# B&R Automation Studio project NAINV104C00R8L515F00 (part 13)

#### Act_EntP0940Disp.st
```iecst
ACTION Act_EntP0940Disp:

	//Access Address
	p_tyC0002FullMask ACCESS ADR(tyP0940CommCtrl.tyFullMaskHide);

	p_tyC0005Main ACCESS ADR(tyCommon.tyMain);

	p_tyC0007Notif ACCESS ADR(tyCommon.tyNotif);

	p_tyC0008MsgBox ACCESS ADR(tyP0940CommCtrl.tyMsgBoxHide);

	p_tyC0009Info ACCESS ADR(tyCommon.tyInfo);

	p_tyC0011Loading ACCESS ADR(tyCommon.tyLoading);

	p_tyP0940CommCtrlUSSMEMA ACCESS ADR(tyP0940CommCtrl.tyUSSMEMA);

	p_tyP0940CommCtrlDSSMEMA ACCESS ADR(tyP0940CommCtrl.tyDSSMEMA);

	p_tyP0940CommCtrlUSSMEMA2 ACCESS ADR(tyP0940CommCtrl.tyUSSMEMA2);

	//Display - Upstream
	fUIInRtStatOff(ADR(tyP0940CommCtrl.tyUSSMEMA.tyLyr.uiRtStat));

	IF p_tyMcParamCurr.tyUSCommSMEMA.eSelection = SMEMASelIPC9851Ext THEN
		fUIInRtStatOff(ADR(tyP0940CommCtrl.tyUSSMEMA.tyBtnUBAStat.uiRtStat));

		IF p_tyMcParamCurr.tyUSCommSMEMA.bStatSigSetGd = TRUE THEN
			tyP0940CommCtrl.tyUSSMEMA.tyBtnUBAStat.usiTxtIdx	:= 1;
		ELSE
			tyP0940CommCtrl.tyUSSMEMA.tyBtnUBAStat.usiTxtIdx	:= 2;
		END_IF
	ELSE
		fUIInRtStatHide(ADR(tyP0940CommCtrl.tyUSSMEMA.tyBtnUBAStat.uiRtStat));
	END_IF

	//Display - Upstream 2
	fUIInRtStatOff(ADR(tyP0940CommCtrl.tyUSSMEMA2.tyLyr.uiRtStat));

	IF p_tyMcParamCurr.tyUSCommSMEMA2.eSelection = SMEMASelIPC9851Ext THEN
		fUIInRtStatOff(ADR(tyP0940CommCtrl.tyUSSMEMA2.tyBtnUBAStat.uiRtStat));

		IF p_tyMcParamCurr.tyUSCommSMEMA2.bStatSigSetGd = TRUE THEN
			tyP0940CommCtrl.tyUSSMEMA2.tyBtnUBAStat.usiTxtIdx	:= 1;
		ELSE
			tyP0940CommCtrl.tyUSSMEMA2.tyBtnUBAStat.usiTxtIdx	:= 2;
		END_IF
	ELSE
		fUIInRtStatHide(ADR(tyP0940CommCtrl.tyUSSMEMA2.tyBtnUBAStat.uiRtStat));
	END_IF

	//Display - Downstream
	fUIInRtStatOff(ADR(tyP0940CommCtrl.tyDSSMEMA.tyLyr.uiRtStat));

	IF p_tyMcParamCurr.tyDSCommSMEMA.eSelection = SMEMASelIPC9851Ext THEN
		fUIInRtStatOff(ADR(tyP0940CommCtrl.tyDSSMEMA.tyBtnDBAStat.uiRtStat));

		IF p_tyMcParamCurr.tyDSCommSMEMA.bStatSigSetGd = TRUE THEN
			tyP0940CommCtrl.tyDSSMEMA.tyBtnDBAStat.usiTxtIdx	:= 1;
		ELSE
			tyP0940CommCtrl.tyDSSMEMA.tyBtnDBAStat.usiTxtIdx	:= 2;
		END_IF
	ELSE
		fUIInRtStatHide(ADR(tyP0940CommCtrl.tyDSSMEMA.tyBtnDBAStat.uiRtStat));
	END_IF

END_ACTION
```

#### Act_OptP0940FullMask.st
```iecst
ACTION Act_OptP0940FullMask:

	IF eCurrPage = UIP0940CommCtrl THEN

		IF p_tyDI.bEStopSig = FALSE THEN
			p_tyC0002FullMask ACCESS ADR(tyP0940CommCtrl.tyFullMaskEStop);

		ELSIF p_tyDI.bCoverSWSig = FALSE THEN
			p_tyC0002FullMask ACCESS ADR(tyP0940CommCtrl.tyFullMaskCWSig);

		ELSIF p_tyDI.bSafetyRlySig = FALSE THEN
			p_tyC0002FullMask ACCESS ADR(tyP0940CommCtrl.tyFullMaskSafetyRly);

		ELSE
			p_tyC0002FullMask ACCESS ADR(tyP0940CommCtrl.tyFullMaskHide);

		END_IF

	END_IF

END_ACTION
```

#### Act_OptP0940ReadDI.st
```iecst
ACTION Act_OptP0940ReadDI:

	tyP0940CommCtrl.tyUSSMEMA.tyBtnUBA.bValue			:= p_tyDI.bUBA;
	tyP0940CommCtrl.tyUSSMEMA.tyBtnUBAStat.bValue		:= p_tyDI.bUBAStat;

	tyP0940CommCtrl.tyDSSMEMA.tyBtnDSB.bValue			:= p_tyDI.bDSB;

	tyP0940CommCtrl.tyUSSMEMA2.tyBtnUBA.bValue			:= p_tyDI.bUBA2;
	tyP0940CommCtrl.tyUSSMEMA2.tyBtnUBAStat.bValue		:= p_tyDI.bUBAStat2;

END_ACTION
```

#### Act_OptP0940WriteDO.st
```iecst
ACTION Act_OptP0940WriteDO:

	// USB
	IF tyP0940CommCtrl.tyUSSMEMA.tyBtnUSB.bRtCompl = TRUE THEN
		IF tyP0940CommCtrl.tyUSSMEMA.tyBtnUSB.bValue = TRUE THEN
			eUSSMEMAAct	:= SMEMAActSetSig;

			IF p_eUSSMEMAStat = SMEMAActSetSig AND p_eUSSMEMAStatus = Done THEN
				eUSSMEMAAct	:= SMEMAActIdle;

				tyP0940CommCtrl.tyUSSMEMA.tyBtnUSB.bRtCompl	:= FALSE;
			END_IF
		ELSE
			eUSSMEMAAct	:= SMEMAActRstSig;

			IF p_eUSSMEMAStat = SMEMAActRstSig AND p_eUSSMEMAStatus = Done THEN
				eUSSMEMAAct	:= SMEMAActIdle;

				tyP0940CommCtrl.tyUSSMEMA.tyBtnUSB.bRtCompl	:= FALSE;
			END_IF
		END_IF
	END_IF

	// USB2
	IF tyP0940CommCtrl.tyUSSMEMA2.tyBtnUSB.bRtCompl = TRUE THEN
		IF tyP0940CommCtrl.tyUSSMEMA2.tyBtnUSB.bValue = TRUE THEN
			eUSSMEMA2Act	:= SMEMAActSetSig;

			IF p_eUSSMEMA2Stat = SMEMAActSetSig AND p_eUSSMEMA2Status = Done THEN
				eUSSMEMA2Act	:= SMEMAActIdle;

				tyP0940CommCtrl.tyUSSMEMA2.tyBtnUSB.bRtCompl	:= FALSE;
			END_IF
		ELSE
			eUSSMEMA2Act	:= SMEMAActRstSig;

			IF p_eUSSMEMA2Stat = SMEMAActRstSig AND p_eUSSMEMA2Status = Done THEN
				eUSSMEMA2Act	:= SMEMAActIdle;

				tyP0940CommCtrl.tyUSSMEMA2.tyBtnUSB.bRtCompl	:= FALSE;
			END_IF
		END_IF
	END_IF

	// DBA
	IF tyP0940CommCtrl.tyDSSMEMA.tyBtnDBA.bRtCompl = TRUE THEN
		IF tyP0940CommCtrl.tyDSSMEMA.tyBtnDBA.bValue = TRUE THEN
			eDSSMEMAAct	:= SMEMAActSetSig;

			IF p_eDSSMEMAStat = SMEMAActSetSig AND p_eDSSMEMAStatus = Done THEN
				eDSSMEMAAct	:= SMEMAActIdle;

				tyP0940CommCtrl.tyDSSMEMA.tyBtnDBA.bRtCompl	:= FALSE;
			END_IF
		ELSE
			eDSSMEMAAct	:= SMEMAActRstSig;

			IF p_eDSSMEMAStat = SMEMAActRstSig AND p_eDSSMEMAStatus = Done THEN
				eDSSMEMAAct	:= SMEMAActIdle;

				tyP0940CommCtrl.tyDSSMEMA.tyBtnDBA.bRtCompl	:= FALSE;
			END_IF
		END_IF
	END_IF

	// DBA Stat
	IF tyP0940CommCtrl.tyDSSMEMA.tyBtnDBAStat.bRtCompl = TRUE THEN
		IF tyP0940CommCtrl.tyDSSMEMA.tyBtnDBAStat.bValue = TRUE THEN
			eDSSMEMAAct	:= SMEMAActSetStatSig;

			IF p_eDSSMEMAStat = SMEMAActSetStatSig AND p_eDSSMEMAStatus = Done THEN
				eDSSMEMAAct	:= SMEMAActIdle;

				tyP0940CommCtrl.tyDSSMEMA.tyBtnDBAStat.bRtCompl	:= FALSE;
			END_IF
		ELSE
			eDSSMEMAAct	:= SMEMAActRstStatSig;

			IF p_eDSSMEMAStat = SMEMAActRstStatSig AND p_eDSSMEMAStatus = Done THEN
				eDSSMEMAAct	:= SMEMAActIdle;

				tyP0940CommCtrl.tyDSSMEMA.tyBtnDBAStat.bRtCompl	:= FALSE;
			END_IF
		END_IF
	END_IF

END_ACTION
```

#### Act_OptP0940UpdtDat.st
```iecst
ACTION Act_OptP0940UpdtDat:

	//Hermes Comm
	//Upstream
	g_tyP0940CommCtrl.tyHermesUS.tyBitmapHermes.uiMaskRtStat.0		:= tyUSHermesBackgndData.bConnectionOK;
	g_tyP0940CommCtrl.tyHermesUS.tyBtnExecute.uiMaskRtStat.0		:= tyUSHermesBackgndData.bConnectionOK;

	IF tyUSHermesBackgndData.bConnectionOK = FALSE THEN
		g_tyP0940CommCtrl.tyHermesUS.tyTxtStat.usiValueIdx	:= 0;
	ELSIF tyUSHermesBackgndData.bConnectionOK = TRUE THEN
		g_tyP0940CommCtrl.tyHermesUS.tyTxtStat.usiValueIdx	:= 1;
	END_IF

	//LED ON
	g_tyP0940CommCtrl.tyHermesUS.tyBtnChkAlive.bValue				:= tyUSHermesBackgndData.tyHermesAllDataFromUS.tyCheckAlive.bChkAlive;
	g_tyP0940CommCtrl.tyHermesUS.tyBtnServiceDescription.bValue		:= tyUSHermesBackgndData.tyHermesAllDataFromUS.tyServiceDescription.bServiceDescription;
	g_tyP0940CommCtrl.tyHermesUS.tyBtnBrdAvl.bValue					:= tyUSHermesBackgndData.tyHermesAllDataFromUS.tyBoardAvailable.bBrdAvl;
	g_tyP0940CommCtrl.tyHermesUS.tyBtnRevokeBrdAvl.bValue			:= tyUSHermesBackgndData.tyHermesAllDataFromUS.tyRevokeBoardAvailable.bRevokeBrdAvl;
	g_tyP0940CommCtrl.tyHermesUS.tyBtnTransportFinished.bValue		:= tyUSHermesBackgndData.tyHermesAllDataFromUS.tyTransportFinished.bTransportFinished;

	//Downstream
	g_tyP0940CommCtrl.tyHermesDS.tyBitmapHermes.uiMaskRtStat.0		:= tyDSHermesBackgndData.bConnectionOK;
	g_tyP0940CommCtrl.tyHermesDS.tyBtnExecute.uiMaskRtStat.0		:= tyDSHermesBackgndData.bConnectionOK;

	IF tyDSHermesBackgndData.bConnectionOK = FALSE THEN
		g_tyP0940CommCtrl.tyHermesDS.tyTxtStat.usiValueIdx	:= 0;
	ELSIF tyDSHermesBackgndData.bConnectionOK = TRUE THEN
		g_tyP0940CommCtrl.tyHermesDS.tyTxtStat.usiValueIdx	:= 1;
	END_IF

	//LED ON
	g_tyP0940CommCtrl.tyHermesDS.tyBtnChkAlive.bValue				:= tyDSHermesBackgndData.tyHermesAllDataFromDS.tyCheckAlive.bChkAlive;
	g_tyP0940CommCtrl.tyHermesDS.tyBtnServiceDescription.bValue		:= tyDSHermesBackgndData.tyHermesAllDataFromDS.tyServiceDescription.bServiceDescription;
	g_tyP0940CommCtrl.tyHermesDS.tyBtnMcRdy.bValue					:= tyDSHermesBackgndData.tyHermesAllDataFromDS.tyMachineReady.bMcRdy;
	g_tyP0940CommCtrl.tyHermesDS.tyBtnRevokeMcRdy.bValue			:= tyDSHermesBackgndData.tyHermesAllDataFromDS.tyRevokeMachineReady.bRevokeMcRdy;
	g_tyP0940CommCtrl.tyHermesDS.tyBtnStartTransport.bValue			:= tyDSHermesBackgndData.tyHermesAllDataFromDS.tyStartTransport.bStartTransport;
	g_tyP0940CommCtrl.tyHermesDS.tyBtnStopTransport.bValue			:= tyDSHermesBackgndData.tyHermesAllDataFromDS.tyStopTransport.bStopTransport;

END_ACTION
```

#### Act_OptP0940MsgCtrl.st
```iecst
ACTION Act_OptP0940MsgCtrl:

	//Upstream
	IF g_tyP0940CommCtrl.tyHermesUS.tyBtnExecute.bRtCompl = TRUE THEN
		g_tyP0940CommCtrl.tyHermesUS.tyBtnExecute.bRtCompl	:= FALSE;
		g_tyP0940CommCtrl.tyHermesUS.tyBtnExecute.bValue	:= FALSE;

		IF g_tyP0940CommCtrl.tyHermesUS.tyDrpDnMsgList.usiValueIdx = 0 THEN
			tyUSHermesBackgndData.tyHermesAllDataToUS.tyCheckAlive.bChkAlive					:= TRUE;
		ELSIF g_tyP0940CommCtrl.tyHermesUS.tyDrpDnMsgList.usiValueIdx = 1 THEN
			tyUSHermesBackgndData.tyHermesAllDataToUS.tyServiceDescription.bServiceDescription	:= TRUE;
		ELSIF g_tyP0940CommCtrl.tyHermesUS.tyDrpDnMsgList.usiValueIdx = 2 THEN
			tyUSHermesBackgndData.tyHermesAllDataToUS.tyMachineReady.bMcRdy						:= TRUE;
		ELSIF g_tyP0940CommCtrl.tyHermesUS.tyDrpDnMsgList.usiValueIdx = 3 THEN
			tyUSHermesBackgndData.tyHermesAllDataToUS.tyRevokeMachineReady.bRevokeMcRdy			:= TRUE;
		ELSIF g_tyP0940CommCtrl.tyHermesUS.tyDrpDnMsgList.usiValueIdx = 4 THEN
			tyUSHermesBackgndData.tyHermesAllDataToUS.tyStartTransport.bStartTransport			:= TRUE;
		ELSIF g_tyP0940CommCtrl.tyHermesUS.tyDrpDnMsgList.usiValueIdx = 5 THEN
			tyUSHermesBackgndData.tyHermesAllDataToUS.tyStopTransport.bStopTransport			:= TRUE;
		ELSIF g_tyP0940CommCtrl.tyHermesUS.tyDrpDnMsgList.usiValueIdx = 6 THEN
			fbUSHermesBackgnd1.eAct	:= HermesBackgroundActIdle;
		END_IF
	END_IF

	//Downstream
	IF g_tyP0940CommCtrl.tyHermesDS.tyBtnExecute.bRtCompl = TRUE THEN
		g_tyP0940CommCtrl.tyHermesDS.tyBtnExecute.bRtCompl	:= FALSE;
		g_tyP0940CommCtrl.tyHermesDS.tyBtnExecute.bValue	:= FALSE;

		IF g_tyP0940CommCtrl.tyHermesDS.tyDrpDnMsgList.usiValueIdx = 0 THEN
			tyDSHermesBackgndData.tyHermesAllDataToDS.tyCheckAlive.bChkAlive					:= TRUE;
		ELSIF g_tyP0940CommCtrl.tyHermesDS.tyDrpDnMsgList.usiValueIdx = 1 THEN
			tyDSHermesBackgndData.tyHermesAllDataToDS.tyServiceDescription.bServiceDescription	:= TRUE;
		ELSIF g_tyP0940CommCtrl.tyHermesDS.tyDrpDnMsgList.usiValueIdx = 2 THEN
			tyDSHermesBackgndData.tyHermesAllDataToDS.tyBoardAvailable.bBrdAvl					:= TRUE;
		ELSIF g_tyP0940CommCtrl.tyHermesDS.tyDrpDnMsgList.usiValueIdx = 3 THEN
			tyDSHermesBackgndData.tyHermesAllDataToDS.tyRevokeBoardAvailable.bRevokeBrdAvl		:= TRUE;
		ELSIF g_tyP0940CommCtrl.tyHermesDS.tyDrpDnMsgList.usiValueIdx = 4 THEN
			tyDSHermesBackgndData.tyHermesAllDataToDS.tyTransportFinished.bTransportFinished	:= TRUE;
		ELSIF g_tyP0940CommCtrl.tyHermesDS.tyDrpDnMsgList.usiValueIdx = 5 THEN
			fbDSHermesBackgnd1.eAct	:= HermesBackgroundActIdle;
		END_IF
	END_IF

END_ACTION
```

#### Act_OptP0940RstMnl.st
```iecst
ACTION Act_OptP0940RstMnl:

	IF EDGEPOS((bManualMod = FALSE) OR (p_eUSSMEMAStatus = Error OR p_eDSSMEMAStatus = Error)) THEN

		eUSSMEMAAct		:= SMEMAActIdle;
		eDSSMEMAAct		:= SMEMAActIdle;
		eUSSMEMA2Act	:= SMEMAActIdle;

		//SMEMA
		tyP0940CommCtrl.tyUSSMEMA.tyBtnUSB.bValue			:= FALSE;
		tyP0940CommCtrl.tyDSSMEMA.tyBtnDBA.bValue			:= FALSE;
		tyP0940CommCtrl.tyDSSMEMA.tyBtnDBAStat.bValue		:= FALSE;
		tyP0940CommCtrl.tyUSSMEMA2.tyBtnUBA.bValue			:= FALSE;

	END_IF

END_ACTION
```

#### Act_EntP0950Disp.st
```iecst
ACTION Act_EntP0950Disp:

	//Access Address
	p_tyC0005Main ACCESS ADR(tyCommon.tyMain);

	p_tyC0007Notif ACCESS ADR(tyCommon.tyNotif);

	p_tyC0008MsgBox ACCESS ADR(tyP0950Simu.tyMsgBoxHide);

	p_tyC0002FullMask ACCESS ADR (tyP0950Simu.tyFullMaskHide);

	p_tyC0009Info ACCESS ADR(tyCommon.tyInfo);

	p_tyP0950Simu ACCESS ADR(tyP0950Simu.tySimu);

	p_tyC0011Loading ACCESS ADR(tyCommon.tyLoading);

END_ACTION
```

#### Act_OptP0950SimulationMod.st
```iecst
ACTION Act_OptP0950SimulationMod:

	IF p_bSimuStatusRun THEN
		tyP0950Simu.tySimu.tyBtnSimu.bRtLk				:= TRUE;
	ELSE
		tyP0950Simu.tySimu.tyBtnSimu.bRtLk				:= tyP0950Simu.tySimu.tyBtnSimu.bValue;
	END_IF

	IF tyP0950Simu.tySimu.tyBtnSimu.bRtCompl THEN
		tyP0950Simu.tySimu.tyBtnSimu.bRtCompl 			:= FALSE;
		tyP0950Simu.tySimu.tyBtnSimu.bValue	  			:= TRUE;
		tyP0950Simu.tySimu.tyBtnSimu.bRtLk	  			:= TRUE;
	END_IF

END_ACTION
```

#### Act_OptP0950Control.st
```iecst
ACTION Act_OptP0950Control:

	// Error
	IF EDGEPOS(p_bAlarmErr = TRUE AND p_bSimuStatusStop = FALSE) THEN

		tyP0950Simu.tySimu.tyBtnStart.bRtCompl	:= FALSE;
		tyP0950Simu.tySimu.tyBtnStop.bRtCompl	:= FALSE;

		tyP0950Simu.tySimu.tyBtnStart.bValue	:= FALSE;
		tyP0950Simu.tySimu.tyBtnStop.bValue		:= FALSE;

		eSimuAct	:= SimulationsActError;

	ELSE

		IF p_eSimuStat = SimulationsActError AND p_eSimuStatus = Done THEN
			eSimuAct	:= SimulationsActIdle;

			bSimuMod	:= FALSE;

		END_IF

	END_IF

	//Control
	IF tyP0950Simu.tySimu.tyBtnStart.bRtCompl = TRUE THEN
		tyP0950Simu.tySimu.tyBtnStop.bRtCompl	:= FALSE;

		eSimuAct		:= SimulationsActStart;

		bSimuMod		:= TRUE;

		IF p_eSimuStat = SimulationsActStart AND p_eSimuStatus = Done THEN
			eSimuAct	:= SimulationsActIdle;

			tyP0950Simu.tySimu.tyBtnStart.bRtCompl	:= FALSE;

		END_IF

	ELSIF tyP0950Simu.tySimu.tyBtnStop.bRtCompl = TRUE THEN
		tyP0950Simu.tySimu.tyBtnStart.bRtCompl	:= FALSE;

		eSimuAct			:= SimulationsActStop;

		IF p_eSimuStat = SimulationsActStop AND p_eSimuStatus = Done THEN
			eSimuAct		:= SimulationsActIdle;
			bSimuMod		:= FALSE;

			tyP0950Simu.tySimu.tyBtnStop.bRtCompl	:= FALSE;
		END_IF

	END_IF

	// Mask
	IF p_bAlarmErr = TRUE THEN
		fUIInRtStatOff(ADR(tyP0950Simu.tySimu.tyBtnStart.uiMaskRtStat));
		fUIInRtStatOff(ADR(tyP0950Simu.tySimu.tyBtnStop.uiMaskRtStat));

	ELSIF p_bSimuStatusCycleStop = TRUE THEN
		fUIInRtStatHide(ADR(tyP0950Simu.tySimu.tyBtnStart.uiMaskRtStat));
		fUIInRtStatOff(ADR(tyP0950Simu.tySimu.tyBtnStop.uiMaskRtStat));

		fbStopBlinkTm(IN := TRUE);
		IF fbStopBlinkTm.Q = TRUE THEN
			fbStopBlinkTm(IN := FALSE);

			tyP0950Simu.tySimu.tyBtnStart.bValue		:= NOT tyP0950Simu.tySimu.tyBtnStart.bValue;
		END_IF

	ELSIF p_bSimuStatusRun = TRUE THEN
		fUIInRtStatOff(ADR(tyP0950Simu.tySimu.tyBtnStart.uiMaskRtStat));
		fUIInRtStatHide(ADR(tyP0950Simu.tySimu.tyBtnStop.uiMaskRtStat));

	ELSE
		fUIInRtStatHide(ADR(tyP0950Simu.tySimu.tyBtnStart.uiMaskRtStat));
		fUIInRtStatOff(ADR(tyP0950Simu.tySimu.tyBtnStop.uiMaskRtStat));

	END_IF

END_ACTION
```

#### Act_EntP1000Disp.st
```iecst
ACTION Act_EntP1000Disp:

	//Access Address
	p_tyC0005Main ACCESS ADR(tyCommon.tyMain);

	p_tyC0007Notif ACCESS ADR(tyCommon.tyNotif);

	p_tyC0008MsgBox ACCESS ADR(tyP1000Lang.tyMsgBoxHide);

	p_tyC0009Info ACCESS ADR(tyCommon.tyInfo);

	p_tyC0011Loading ACCESS ADR(tyCommon.tyLoading);

	p_tyP1000Lang ACCESS ADR(tyP1000Lang.tyLang);

	//Backup Param
	tyP1000Lang.tyLangBkUp	:= tyP1000Lang.tyLang;

	//Display
	tyP1000Lang.tyLang.tyBtnEnglish.uiRtStat.0		:= NOT (p_tyNtParamCurr.bChinesePrep OR p_tyNtParamCurr.bGemanPrep);
	tyP1000Lang.tyLang.tyBtnChinese.uiRtStat.0		:= NOT (p_tyNtParamCurr.bChinesePrep);
	tyP1000Lang.tyLang.tyBtnGerman.uiRtStat.0		:= NOT (p_tyNtParamCurr.bGemanPrep);

END_ACTION
```

#### Act_ExitP1000.st
```iecst
ACTION Act_ExitP1000:

	eMcParamAct	:= McParamActWrite;

	IF p_eMcParamStat = McParamActWrite AND p_eMcParamStatus = Done THEN
		eMcParamAct	:= McParamActIdle;

		usiChgPage	:= 1;

	ELSIF p_eMcParamStatus = Error THEN
		p_tyC0008MsgBox ACCESS ADR(tyP1000Lang.tyMsgBoxSaveErr);

		IF tyP1000Lang.tyMsgBoxSaveErr.tyBtnNo.bRtCompl = TRUE THEN
			tyP1000Lang.tyMsgBoxSaveErr.tyBtnNo.bRtCompl	:= FALSE;
			tyP1000Lang.tyMsgBoxSaveErr.tyBtnNo.bValue		:= FALSE;

			p_tyC0008MsgBox ACCESS ADR(tyP1000Lang.tyMsgBoxHide);

			//Restore Param
			tyP1000Lang.tyLang				:= tyP1000Lang.tyLangBkUp;
			tyMcParamWr						:= p_tyMcParamCurr;
			tyProperty.tyVisu.usiChgLang	:= p_tyMcParamCurr.usiLang;

			usiChgPage	:= 1;

		END_IF

	END_IF

END_ACTION
```

#### Act_OptP1000SelectLang.st
```iecst
ACTION Act_OptP1000SelectLang:

	// Select English Language
	IF tyP1000Lang.tyLang.tyBtnEnglish.bRtCompl = TRUE THEN
		tyP1000Lang.tyLang.tyBtnEnglish.bRtCompl	:= FALSE;

		tyP1000Lang.tyLang.tyBtnEnglish.bValue		:= TRUE;
		tyP1000Lang.tyLang.tyBtnGerman.bValue		:= FALSE;
		tyP1000Lang.tyLang.tyBtnChinese.bValue		:= FALSE;

		tyP1000Lang.tyLang.tyBtnEnglish.bRtLk		:= TRUE;
		tyP1000Lang.tyLang.tyBtnGerman.bRtLk		:= FALSE;
		tyP1000Lang.tyLang.tyBtnChinese.bRtLk		:= FALSE;

		tyProperty.tyVisu.usiChgLang	:= 0;

		tyMcParamWr.usiLang	:= 0;

	// Select German Language
	ELSIF tyP1000Lang.tyLang.tyBtnGerman.bRtCompl = TRUE THEN
		tyP1000Lang.tyLang.tyBtnGerman.bRtCompl	:= FALSE;

		tyP1000Lang.tyLang.tyBtnEnglish.bValue	:= FALSE;
		tyP1000Lang.tyLang.tyBtnGerman.bValue	:= TRUE;
		tyP1000Lang.tyLang.tyBtnChinese.bValue	:= FALSE;

		tyP1000Lang.tyLang.tyBtnEnglish.bRtLk	:= FALSE;
		tyP1000Lang.tyLang.tyBtnGerman.bRtLk	:= TRUE;
		tyP1000Lang.tyLang.tyBtnChinese.bRtLk	:= FALSE;

		tyProperty.tyVisu.usiChgLang	:= 1;

		tyMcParamWr.usiLang	:= 1;

	// Select Chinese Language
	ELSIF tyP1000Lang.tyLang.tyBtnChinese.bRtCompl = TRUE THEN
		tyP1000Lang.tyLang.tyBtnChinese.bRtCompl	:= FALSE;

		tyP1000Lang.tyLang.tyBtnEnglish.bValue		:= FALSE;
		tyP1000Lang.tyLang.tyBtnGerman.bValue		:= FALSE;
		tyP1000Lang.tyLang.tyBtnChinese.bValue		:= TRUE;

		tyP1000Lang.tyLang.tyBtnEnglish.bRtLk		:= FALSE;
		tyP1000Lang.tyLang.tyBtnGerman.bRtLk		:= FALSE;
		tyP1000Lang.tyLang.tyBtnChinese.bRtLk		:= TRUE;

		tyProperty.tyVisu.usiChgLang	:= 2;

		tyMcParamWr.usiLang	:= 2;

	END_IF

END_ACTION
```

#### Act_OptP1000Keypad.st
```iecst
ACTION Act_OptP1000Keypad:

	IF fUIOutRtStatTPIsOpen(ADR(tyP1000Lang.tyLang.tyNumDay.uiRtStat)) = TRUE THEN
		tyProperty.tyKeypad.tyTxtTitle.sTxt			:= tyP1000Lang.tyLang.tyNumDay.sKeypadTitle;

	ELSIF fUIOutRtStatTPIsOpen(ADR(tyP1000Lang.tyLang.tyNumMonth.uiRtStat)) = TRUE THEN
		tyProperty.tyKeypad.tyTxtTitle.sTxt			:= tyP1000Lang.tyLang.tyNumMonth.sKeypadTitle;

	ELSIF fUIOutRtStatTPIsOpen(ADR(tyP1000Lang.tyLang.tyNumYear.uiRtStat)) = TRUE THEN
		tyProperty.tyKeypad.tyTxtTitle.sTxt			:= tyP1000Lang.tyLang.tyNumYear.sKeypadTitle;

	ELSIF fUIOutRtStatTPIsOpen(ADR(tyP1000Lang.tyLang.tyNumSecond.uiRtStat)) = TRUE THEN
		tyProperty.tyKeypad.tyTxtTitle.sTxt			:= tyP1000Lang.tyLang.tyNumSecond.sKeypadTitle;

	ELSIF fUIOutRtStatTPIsOpen(ADR(tyP1000Lang.tyLang.tyNumMinute.uiRtStat)) = TRUE THEN
		tyProperty.tyKeypad.tyTxtTitle.sTxt			:= tyP1000Lang.tyLang.tyNumMinute.sKeypadTitle;

	ELSIF fUIOutRtStatTPIsOpen(ADR(tyP1000Lang.tyLang.tyNumHour.uiRtStat)) = TRUE THEN
		tyProperty.tyKeypad.tyTxtTitle.sTxt			:= tyP1000Lang.tyLang.tyNumHour.sKeypadTitle;

	END_IF

END_ACTION
```

#### Act_EntP1020Disp.st
```iecst
ACTION Act_EntP1020Disp:

	//Access Address
	p_tyC0005Main ACCESS ADR(tyCommon.tyMain);

	p_tyC0007Notif ACCESS ADR(tyCommon.tyNotif);

	p_tyC0008MsgBox ACCESS ADR(tyP1020McSetNavi.tyMsgBoxHide);

	p_tyC0009Info ACCESS ADR(tyCommon.tyInfo);

	p_tyC0011Loading ACCESS ADR(tyCommon.tyLoading);

	p_tyP1020McSetNavi ACCESS ADR(tyP1020McSetNavi.tyNavi);

END_ACTION
```

#### Act_OptP1020Navi.st
```iecst
ACTION Act_OptP1020Navi:

	IF tyP1020McSetNavi.tyNavi.tyBtnMcSet.bRtCompl = TRUE THEN
		tyP1020McSetNavi.tyNavi.tyBtnMcSet.bRtCompl	:= FALSE;
		tyP1020McSetNavi.tyNavi.tyBtnMcSet.bValue	:= FALSE;

		eChgPage	:= UIP1021McSetGen;

	ELSIF tyP1020McSetNavi.tyNavi.tyBtnVCommSet.bRtCompl = TRUE THEN
		tyP1020McSetNavi.tyNavi.tyBtnVCommSet.bRtCompl	:= FALSE;
		tyP1020McSetNavi.tyNavi.tyBtnVCommSet.bValue	:= FALSE;

		eChgPage	:= UIP1022McSetVComm;

	ELSIF tyP1020McSetNavi.tyNavi.tyBtnHCommSet.bRtCompl = TRUE THEN
		tyP1020McSetNavi.tyNavi.tyBtnHCommSet.bRtCompl	:= FALSE;
		tyP1020McSetNavi.tyNavi.tyBtnHCommSet.bValue	:= FALSE;

		eChgPage	:= UIP1023McSetHComm;

	ELSIF tyP1020McSetNavi.tyNavi.tyBtnAntiGapSet.bRtCompl = TRUE THEN
		tyP1020McSetNavi.tyNavi.tyBtnAntiGapSet.bRtCompl	:= FALSE;
		tyP1020McSetNavi.tyNavi.tyBtnAntiGapSet.bValue		:= FALSE;

		eChgPage	:= UIP1024McSetAntiGap;

	END_IF

END_ACTION
```

#### Act_EntP1021McSetDisp.st
```iecst
ACTION Act_EntP1021Disp:

	//Access Address
	IF bTeachStopperAtLftPos = TRUE OR bTeachStopperAtRgtPos = TRUE THEN
		p_tyC0004Navi ACCESS ADR(tyP1021McSetGen.tyNaviLyr2);
	ELSE
		p_tyC0004Navi ACCESS ADR(tyP1021McSetGen.tyNaviLyr1);
	END_IF

	p_tyC0005Main ACCESS ADR(tyCommon.tyMain);

	p_tyC0006Set ACCESS ADR(tyCommon.tySet);

	p_tyC0007Notif ACCESS ADR(tyCommon.tyNotif);

	p_tyC0008MsgBox ACCESS ADR(tyP1021McSetGen.tyMsgBoxHide);

	p_tyC0009Info ACCESS ADR(tyCommon.tyInfo);

	p_tyC0011Loading ACCESS ADR(tyCommon.tyLoading);

	p_tyP1021McSetGen ACCESS ADR(tyP1021McSetGen.tyGen);

	p_tyP1021McSetNetwork ACCESS ADR(tyP1021McSetGen.tyNetwork);
	//Display
	tyP1021McSetGen.tyGen.tyLyrGen1.uiRtStat.0	:= bTeachStopperAtLftPos OR bTeachStopperAtRgtPos;
	tyP1021McSetGen.tyGen.tyLyrGen2.uiRtStat.0	:= NOT(bTeachStopperAtLftPos OR bTeachStopperAtRgtPos);

	//Backup Param
	IF NOT(bTeachStopperAtLftPos OR bTeachStopperAtRgtPos) THEN
		tyP1021McSetGen.tyGenBkUp	:= tyP1021McSetGen.tyGen;
	ELSE
		bTeachStopperAtLftPos	:= FALSE;
		bTeachStopperAtRgtPos	:= FALSE;
	END_IF

	//Network Configuration Display
	usiNetworkModeOld := DINT_TO_USINT(p_tyMcParamCurr.eNetworkMod);

	fUIInRtStatHide(ADR(tyP1021McSetGen.tyNetwork.tyLyr.uiRtStat));

	tyP1021McSetGen.tyGen.tyBtnLFBuzMute.uiRtStat.0 := NOT (p_tyMcParamCurr.bLFEn AND p_tyNtParamCurr.bLFPrep AND p_tyNtParamCurr.tyDOSettings.diBuz > 0);
END_ACTION
```

#### Act_ExitP1021.st
```iecst
ACTION Act_ExitP1021:

	IF tyCommon.tySet.tyBtnSave.uiMaskRtStat.0 = FALSE THEN
		usiChgPage	:= 1;

	ELSE
		p_tyC0008MsgBox ACCESS ADR(tyP1021McSetGen.tyMsgBoxExitAsk);

		IF tyP1021McSetGen.tyMsgBoxExitAsk.tyBtnYes.bRtCompl = TRUE THEN
			tyP1021McSetGen.tyMsgBoxExitAsk.tyBtnYes.bRtCompl	:= FALSE;
			tyP1021McSetGen.tyMsgBoxExitAsk.tyBtnYes.bValue		:= FALSE;

			p_tyC0008MsgBox ACCESS ADR(tyP1021McSetGen.tyMsgBoxHide);

			//Recover Param
			tyP1021McSetGen.tyGen	:= tyP1021McSetGen.tyGenBkUp;

			fUIInRtStatOff(ADR(tyCommon.tySet.tyBtnSave.uiMaskRtStat));

			bSaveNetworkPriority	:= FALSE;

			usiChgPage	:= 1;

		ELSIF tyP1021McSetGen.tyMsgBoxExitAsk.tyBtnNo.bRtCompl = TRUE THEN
			tyP1021McSetGen.tyMsgBoxExitAsk.tyBtnNo.bRtCompl	:= FALSE;
			tyP1021McSetGen.tyMsgBoxExitAsk.tyBtnNo.bValue		:= FALSE;

			p_tyC0008MsgBox ACCESS ADR(tyP1021McSetGen.tyMsgBoxHide);

			eChgPage	:= eCurrPage;
			usiChgPage	:= 0;

		END_IF

	END_IF

END_ACTION
```

#### Act_OptP1021Navi.st
```iecst
ACTION Act_OptP1021Navi:

	IF tyP1021McSetGen.tyNaviLyr1.tyBtnBack.bRtCompl = TRUE OR tyP1021McSetGen.tyNaviLyr2.tyBtnBack.bRtCompl = TRUE THEN
		eChgPage	:= UIP1020McSetNavi;

		tyP1021McSetGen.tyNaviLyr1.tyBtnBack.bRtCompl	:= FALSE;
		tyP1021McSetGen.tyNaviLyr2.tyBtnBack.bRtCompl	:= FALSE;

	//Navi From Layer 1 to Layer 2
	ELSIF tyP1021McSetGen.tyNaviLyr1.tyBtnRgt.bRtCompl = TRUE THEN
		p_tyC0004Navi ACCESS ADR (tyP1021McSetGen.tyNaviLyr2);

		fUIInRtStatHide(ADR(tyP1021McSetGen.tyGen.tyLyrGen1.uiRtStat));
		fUIInRtStatOff(ADR(tyP1021McSetGen.tyGen.tyLyrGen2.uiRtStat));

		tyP1021McSetGen.tyNaviLyr1.tyBtnRgt.bRtCompl	:= FALSE;

	ELSIF tyP1021McSetGen.tyNaviLyr1.tyBtnLeft.bRtCompl = TRUE THEN
		p_tyC0004Navi ACCESS ADR (tyP1021McSetGen.tyNaviLyr2);

		fUIInRtStatHide(ADR(tyP1021McSetGen.tyGen.tyLyrGen1.uiRtStat));
		fUIInRtStatOff(ADR(tyP1021McSetGen.tyGen.tyLyrGen2.uiRtStat));

		tyP1021McSetGen.tyNaviLyr1.tyBtnLeft.bRtCompl	:= FALSE;

	//Navi Form Layer 2 to Layer 1
	ELSIF tyP1021McSetGen.tyNaviLyr2.tyBtnRgt.bRtCompl = TRUE THEN
		p_tyC0004Navi ACCESS ADR(tyP1021McSetGen.tyNaviLyr1);

		fUIInRtStatOff(ADR(tyP1021McSetGen.tyGen.tyLyrGen1.uiRtStat));
		fUIInRtStatHide(ADR(tyP1021McSetGen.tyGen.tyLyrGen2.uiRtStat));

		tyP1021McSetGen.tyNaviLyr2.tyBtnRgt.bRtCompl	:= FALSE;

	ELSIF tyP1021McSetGen.tyNaviLyr2.tyBtnLeft.bRtCompl = TRUE THEN
		p_tyC0004Navi ACCESS ADR(tyP1021McSetGen.tyNaviLyr1);

		fUIInRtStatOff(ADR(tyP1021McSetGen.tyGen.tyLyrGen1.uiRtStat));
		fUIInRtStatHide(ADR(tyP1021McSetGen.tyGen.tyLyrGen2.uiRtStat));

		tyP1021McSetGen.tyNaviLyr2.tyBtnLeft.bRtCompl	:= FALSE;

	END_IF

END_ACTION
```

#### Act_OptP1021Save.st
```iecst
ACTION Act_OptP1021Save:

	IF tyP1021McSetGen.tyGen.tyStringMcNm.bRtCompl 					OR tyP1021McSetGen.tyGen.tyDrpDnDefaultMcMod.bRtCompl
		OR tyP1021McSetGen.tyGen.tyDrpDnDefaultFlippedBrd.bRtCompl 	OR tyP1021McSetGen.tyGen.tyNumSSaverTm.bRtCompl
		OR tyP1021McSetGen.tyGen.tyBtnSSaverEn.bRtCompl				OR tyP1021McSetGen.tyGen.tyNumWidthAtHm.bRtCompl
		OR tyP1021McSetGen.tyGen.tyNumConvInitTm.bRtCompl			OR tyP1021McSetGen.tyGen.tyNumTranInErrDlyTm.bRtCompl
		OR tyP1021McSetGen.tyGen.tyNumTranOutErrDlyTm.bRtCompl

		OR tyP1021McSetGen.tyGen.tyBtnAWDis.bRtCompl 				OR tyP1021McSetGen.tyGen.tyBtnVSMEMAEn.bRtCompl
		OR tyP1021McSetGen.tyGen.tyBtnHermesRmtEn.bRtCompl			OR tyP1021McSetGen.tyGen.tyBtnMnlAccDat.bRtCompl
		OR tyP1021McSetGen.tyGen.tyBtnAutoStepEn.bRtCompl			OR tyP1021McSetGen.tyGen.tyBtnChgParamEn.bRtCompl
		OR tyP1021McSetGen.tyGen.tyNumStopperAtLftPos.bRtCompl 		OR tyP1021McSetGen.tyGen.tyNumStopperAtRgtPos.bRtCompl
		OR tyP1021McSetGen.tyGen.tyBtnStopperDis.bRtCompl 		 	OR tyP1021McSetGen.tyGen.tyNumWidthOffset.bRtCompl
		OR tyP1021McSetGen.tyGen.tyBtnAutoLogoutEn.bRtCompl 		OR tyP1021McSetGen.tyGen.tyBtnClampDis.bRtCompl
		OR tyP1021McSetGen.tyGen.tyBtnLFBuzMute.bRtCompl			OR tyP1021McSetGen.tyGen.tyNumAutoLogoutTm.bRtCompl
		THEN

		fUIInRtStatHide(ADR(tyCommon.tySet.tyBtnSave.uiMaskRtStat));

		tyP1021McSetGen.tyGen.tyStringMcNm.bRtCompl 			:= FALSE;
		tyP1021McSetGen.tyGen.tyDrpDnDefaultMcMod.bRtCompl		:= FALSE;
		tyP1021McSetGen.tyGen.tyDrpDnDefaultFlippedBrd.bRtCompl	:= FALSE;
		tyP1021McSetGen.tyGen.tyNumSSaverTm.bRtCompl			:= FALSE;
		tyP1021McSetGen.tyGen.tyBtnSSaverEn.bRtCompl			:= FALSE;
		tyP1021McSetGen.tyGen.tyNumWidthAtHm.bRtCompl			:= FALSE;
		tyP1021McSetGen.tyGen.tyNumWidthOffset.bRtCompl			:= FALSE;
		tyP1021McSetGen.tyGen.tyNumConvInitTm.bRtCompl			:= FALSE;
		tyP1021McSetGen.tyGen.tyNumTranInErrDlyTm.bRtCompl		:= FALSE;
		tyP1021McSetGen.tyGen.tyNumTranOutErrDlyTm.bRtCompl		:= FALSE;

		tyP1021McSetGen.tyGen.tyBtnAWDis.bRtCompl 				:= FALSE;
		tyP1021McSetGen.tyGen.tyBtnVSMEMAEn.bRtCompl			:= FALSE;
		tyP1021McSetGen.tyGen.tyBtnHermesRmtEn.bRtCompl			:= FALSE;
		tyP1021McSetGen.tyGen.tyBtnMnlAccDat.bRtCompl			:= FALSE;
		tyP1021McSetGen.tyGen.tyBtnAutoStepEn.bRtCompl			:= FALSE;
		tyP1021McSetGen.tyGen.tyBtnChgParamEn.bRtCompl			:= FALSE;

		tyP1021McSetGen.tyGen.tyBtnStopperDis.bRtCompl			:= FALSE;
		tyP1021McSetGen.tyGen.tyNumStopperAtLftPos.bRtCompl		:= FALSE;
		tyP1021McSetGen.tyGen.tyNumStopperAtRgtPos.bRtCompl		:= FALSE;
		tyP1021McSetGen.tyGen.tyBtnAutoLogoutEn.bRtCompl		:= FALSE;
		tyP1021McSetGen.tyGen.tyBtnClampDis.bRtCompl			:= FALSE;
		tyP1021McSetGen.tyGen.tyBtnLFBuzMute.bRtCompl			:= FALSE;
		tyP1021McSetGen.tyGen.tyNumAutoLogoutTm.bRtCompl		:= FALSE;

	END_IF

	IF tyCommon.tySet.tyBtnSave.bRtCompl = TRUE AND bSaveNetworkPriority=FALSE THEN
		//Save Param
		tyMcParamWr.sMcNm					:= tyP1021McSetGen.tyGen.tyStringMcNm.sValue;
		tyMcParamWr.usiDefaultMcMod			:= tyP1021McSetGen.tyGen.tyDrpDnDefaultMcMod.usiValueIdx;
		tyMcParamWr.usiDefaultFlippedBrd	:= tyP1021McSetGen.tyGen.tyDrpDnDefaultFlippedBrd.usiValueIdx;
		tyMcParamWr.uiSSaverTmInSec			:= DINT_TO_UINT(tyP1021McSetGen.tyGen.tyNumSSaverTm.diValue);
		tyMcParamWr.bSSaverEn				:= tyP1021McSetGen.tyGen.tyBtnSSaverEn.bValue;
		tyMcParamWr.diAutoLogoutTmInSec		:= tyP1021McSetGen.tyGen.tyNumAutoLogoutTm.diValue;
		tyMcParamWr.bAutoLogoutEn			:= tyP1021McSetGen.tyGen.tyBtnAutoLogoutEn.bValue;
		tyMcParamWr.diWidthAtHmPosInUM		:= tyP1021McSetGen.tyGen.tyNumWidthAtHm.diValue;
		tyMcParamWr.diConvInitTmInMS		:= tyP1021McSetGen.tyGen.tyNumConvInitTm.diValue;
		tyMcParamWr.diTranInErrDlyTmInMS	:= tyP1021McSetGen.tyGen.tyNumTranInErrDlyTm.diValue;
		tyMcParamWr.diTranOutErrDlyTmInMS	:= tyP1021McSetGen.tyGen.tyNumTranOutErrDlyTm.diValue;

		tyMcParamWr.bAWDis					:= tyP1021McSetGen.tyGen.tyBtnAWDis.bValue;
		tyMcParamWr.bVSMEMAEn				:= tyP1021McSetGen.tyGen.tyBtnVSMEMAEn.bValue;
		tyMcParamWr.bHermesRmtEn			:= tyP1021McSetGen.tyGen.tyBtnHermesRmtEn.bValue;
		tyMcParamWr.bMnlAccDat				:= tyP1021McSetGen.tyGen.tyBtnMnlAccDat.bValue;
		tyMcParamWr.bAutoStepEn				:= tyP1021McSetGen.tyGen.tyBtnAutoStepEn.bValue;
		tyMcParamWr.bChgParamEn				:= tyP1021McSetGen.tyGen.tyBtnChgParamEn.bValue;

		tyMcParamWr.bStopperDis				:= tyP1021McSetGen.tyGen.tyBtnStopperDis.bValue;
		tyMcParamWr.diStopperAtLftPos		:= tyP1021McSetGen.tyGen.tyNumStopperAtLftPos.diValue;
		tyMcParamWr.diStopperAtRgtPos		:= tyP1021McSetGen.tyGen.tyNumStopperAtRgtPos.diValue;
		tyMcParamWr.diWidthOffsetInUM		:= tyP1021McSetGen.tyGen.tyNumWidthOffset.diValue;

		tyMcParamWr.bClampDis				:= tyP1021McSetGen.tyGen.tyBtnClampDis.bValue;

		tyMcParamWr.eNetworkMod				:= USINT_TO_DINT(tyP1021McSetGen.tyGen.tyDrpDnNetworkMod.usiValueIdx);

		tyMcParamWr.bLFBuzMute				:= tyP1021McSetGen.tyGen.tyBtnLFBuzMute.bValue;

		IF tyP1021McSetGen.tyGen.tyDrpDnNetworkMod.usiValueIdx =DINT_TO_USINT(SetIPManually) THEN
			tyMcParamWr.sIPAddr				:= tyP1021McSetGen.tyGen.tyStringIPAddr.sValue;
			tyMcParamWr.sSubnetMask			:= tyP1021McSetGen.tyGen.tyStringSubnetMask.sValue;
		END_IF

		eMcParamAct	:= McParamActWrite;

		IF p_eMcParamStat = McParamActWrite AND p_eMcParamStatus = Done THEN
			eMcParamAct	:= McParamActIdle;

			usiNetworkModeOld := tyP1021McSetGen.tyGen.tyDrpDnNetworkMod.usiValueIdx;
			//Update Screen Saver Time
			tyProperty.tyVisu.uiSSaverTm	:= p_tyMcParamCurr.uiSSaverTmInSec;

			//Backup Param
			tyP1021McSetGen.tyGenBkUp	:= tyP1021McSetGen.tyGen;

			tyCommon.tySet.tyBtnSave.bRtCompl	:= FALSE;

			fUIInRtStatOff(ADR(tyCommon.tySet.tyBtnSave.uiMaskRtStat));

		ELSIF p_eMcParamStatus = Error THEN
			p_tyC0008MsgBox ACCESS ADR(tyP1021McSetGen.tyMsgBoxSaveErr);

			IF tyP1021McSetGen.tyMsgBoxSaveErr.tyBtnNo.bRtCompl = TRUE THEN
				tyP1021McSetGen.tyMsgBoxSaveErr.tyBtnNo.bRtCompl	:= FALSE;
				tyP1021McSetGen.tyMsgBoxSaveErr.tyBtnNo.bValue		:= FALSE;

				p_tyC0008MsgBox ACCESS ADR(tyP1021McSetGen.tyMsgBoxHide);

				//Restore Param
				tyP1021McSetGen.tyGen	:= tyP1021McSetGen.tyGenBkUp;
				tyMcParamWr				:= p_tyMcParamCurr;

				tyCommon.tySet.tyBtnSave.bRtCompl	:= FALSE;

				fUIInRtStatOff(ADR(tyCommon.tySet.tyBtnSave.uiMaskRtStat));

			END_IF

		END_IF

	ELSIF bUpdateP1021Network THEN
		tyMcParamWr.sIPAddr					:= tyP1021McSetGen.tyGen.tyStringIPAddr.sValue;
		tyMcParamWr.sSubnetMask				:= tyP1021McSetGen.tyGen.tyStringSubnetMask.sValue;

		eMcParamAct	:= McParamActWrite;

		IF p_eMcParamStat = McParamActWrite AND p_eMcParamStatus = Done THEN
			eMcParamAct		:= McParamActIdle;

			IF bUpdateP1021Network THEN
				bUpdateP1021Network :=FALSE;
			END_IF

			//Update Restore Param
			tyP1021McSetGen.tyGenBkUp.tyStringIPAddr.sValue	 	:= tyP1021McSetGen.tyGen.tyStringIPAddr.sValue;
			tyP1021McSetGen.tyGenBkUp.tyStringSubnetMask.sValue	:= tyP1021McSetGen.tyGen.tyStringSubnetMask.sValue;

		ELSIF p_eMcParamStatus = Error THEN
			p_tyC0008MsgBox ACCESS ADR(tyP1021McSetGen.tyMsgBoxSaveErr);

			IF tyP1021McSetGen.tyMsgBoxSaveErr.tyBtnNo.bRtCompl = TRUE THEN
				tyP1021McSetGen.tyMsgBoxSaveErr.tyBtnNo.bRtCompl 			:= FALSE;
				tyP1021McSetGen.tyMsgBoxSaveErr.tyBtnNo.bValue				:= FALSE;

				p_tyC0008MsgBox ACCESS ADR(tyP1021McSetGen.tyMsgBoxHide);

				// Restore Param
				tyP1021McSetGen.tyGenBkUp.tyStringIPAddr.sValue	 	:= tyP1021McSetGen.tyGen.tyStringIPAddr.sValue;
				tyP1021McSetGen.tyGenBkUp.tyStringSubnetMask.sValue	:= tyP1021McSetGen.tyGen.tyStringSubnetMask.sValue;

				tyMcParamWr				:= p_tyMcParamCurr;

				bUpdateP1021Network :=FALSE;

			END_IF
		END_IF

	END_IF

END_ACTION
```

#### Act_OptP1021Keypad.st
```iecst
ACTION Act_OptP1021Keypad:

	IF fUIOutRtStatTPIsOpen(ADR(tyP1021McSetGen.tyGen.tyStringMcNm.uiRtStat)) = TRUE THEN
		tyProperty.tyKeypad.tyTxtTitle.sTxt	:= tyP1021McSetGen.tyGen.tyStringMcNm.sKeypadTitle;

	ELSIF fUIOutRtStatTPIsOpen(ADR(tyP1021McSetGen.tyGen.tyNumSSaverTm.uiRtStat)) = TRUE THEN
		tyProperty.tyKeypad.tyTxtTitle.sTxt	:= tyP1021McSetGen.tyGen.tyNumSSaverTm.sKeypadTitle;

	ELSIF fUIOutRtStatTPIsOpen(ADR(tyP1021McSetGen.tyGen.tyStringIPAddr.uiRtStat)) = TRUE THEN
		tyProperty.tyKeypad.tyTxtTitle.sTxt	:= tyP1021McSetGen.tyGen.tyStringIPAddr.sKeypadTitle;

	ELSIF fUIOutRtStatTPIsOpen(ADR(tyP1021McSetGen.tyGen.tyStringSubnetMask.uiRtStat)) = TRUE THEN
		tyProperty.tyKeypad.tyTxtTitle.sTxt	:= tyP1021McSetGen.tyGen.tyStringSubnetMask.sKeypadTitle;

	ELSIF fUIOutRtStatTPIsOpen(ADR(tyP1021McSetGen.tyGen.tyNumWidthAtHm.uiRtStat)) = TRUE THEN
		tyProperty.tyKeypad.tyTxtTitle.sTxt	:= tyP1021McSetGen.tyGen.tyNumWidthAtHm.sKeypadTitle;

	ELSIF fUIOutRtStatTPIsOpen(ADR(tyP1021McSetGen.tyGen.tyNumWidthOffset.uiRtStat)) = TRUE THEN
		tyProperty.tyKeypad.tyTxtTitle.sTxt	:= tyP1021McSetGen.tyGen.tyNumWidthOffset.sKeypadTitle;

	ELSIF fUIOutRtStatTPIsOpen(ADR(tyP1021McSetGen.tyGen.tyNumConvInitTm.uiRtStat)) = TRUE THEN
		tyProperty.tyKeypad.tyTxtTitle.sTxt	:= tyP1021McSetGen.tyGen.tyNumConvInitTm.sKeypadTitle;

	ELSIF fUIOutRtStatTPIsOpen(ADR(tyP1021McSetGen.tyGen.tyNumTranInErrDlyTm.uiRtStat)) = TRUE THEN
		tyProperty.tyKeypad.tyTxtTitle.sTxt	:= tyP1021McSetGen.tyGen.tyNumTranInErrDlyTm.sKeypadTitle;

	ELSIF fUIOutRtStatTPIsOpen(ADR(tyP1021McSetGen.tyGen.tyNumTranOutErrDlyTm.uiRtStat)) = TRUE THEN
		tyProperty.tyKeypad.tyTxtTitle.sTxt	:= tyP1021McSetGen.tyGen.tyNumTranOutErrDlyTm.sKeypadTitle;

	ELSIF fUIOutRtStatTPIsOpen(ADR(tyP1021McSetGen.tyGen.tyNumStopperAtLftPos.uiRtStat)) = TRUE THEN
		tyProperty.tyKeypad.tyTxtTitle.sTxt	:= tyP1021McSetGen.tyGen.tyNumStopperAtLftPos.sKeypadTitle;

	ELSIF fUIOutRtStatTPIsOpen(ADR(tyP1021McSetGen.tyGen.tyNumStopperAtRgtPos.uiRtStat)) = TRUE THEN
		tyProperty.tyKeypad.tyTxtTitle.sTxt	:= tyP1021McSetGen.tyGen.tyNumStopperAtRgtPos.sKeypadTitle;

	ELSIF fUIOutRtStatTPIsOpen(ADR(tyP1021McSetGen.tyNetwork.tyStringIPAddr.uiRtStat)) = TRUE THEN
		tyProperty.tyKeypad.tyTxtTitle.sTxt	:= tyP1021McSetGen.tyNetwork.tyStringIPAddr.sKeypadTitle;

	ELSIF fUIOutRtStatTPIsOpen(ADR(tyP1021McSetGen.tyNetwork.tyStringSubnetMask.uiRtStat)) = TRUE THEN
		tyProperty.tyKeypad.tyTxtTitle.sTxt	:= tyP1021McSetGen.tyNetwork.tyStringSubnetMask.sKeypadTitle;

	END_IF

END_ACTION
```

#### Act_OptP1021IPAddr.st
```iecst
ACTION Act_OptP1021IPAddr:

	IF tyP1021McSetGen.tyGen.tyStringIPAddr.bRtCompl = TRUE THEN

		IF fIPValid(tyP1021McSetGen.tyGen.tyStringIPAddr.sValue , ADR(a_iIPPart1)) THEN

			IF usiSaveIPAddrStep = 0 THEN
				p_tyC0008MsgBox ACCESS ADR(tyP1021McSetGen.tyMsgBoxUpdtIPAddrAsk);

				IF tyP1021McSetGen.tyMsgBoxUpdtIPAddrAsk.tyBtnYes.bRtCompl = TRUE THEN
					tyP1021McSetGen.tyMsgBoxUpdtIPAddrAsk.tyBtnYes.bRtCompl	:= FALSE;
					tyP1021McSetGen.tyMsgBoxUpdtIPAddrAsk.tyBtnYes.bValue	:= FALSE;

					p_tyC0008MsgBox ACCESS ADR(tyP1021McSetGen.tyMsgBoxHide);

					usiSaveIPAddrStep	:= 1;

				ELSIF tyP1021McSetGen.tyMsgBoxUpdtIPAddrAsk.tyBtnNo.bRtCompl = TRUE THEN
					tyP1021McSetGen.tyMsgBoxUpdtIPAddrAsk.tyBtnNo.bRtCompl	:= FALSE;
					tyP1021McSetGen.tyMsgBoxUpdtIPAddrAsk.tyBtnNo.bValue	:= FALSE;

					//Recover IP Address
					tyP1021McSetGen.tyGen.tyStringIPAddr.sValue	:= p_sHWInfoIPAddr;

					tyP1021McSetGen.tyGen.tyStringIPAddr.bRtCompl	:= FALSE;

					p_tyC0008MsgBox ACCESS ADR(tyP1021McSetGen.tyMsgBoxHide);

				END_IF

			ELSIF usiSaveIPAddrStep = 1 THEN
				//Set IP Address
				sSetIPAddr	:= tyP1021McSetGen.tyGen.tyStringIPAddr.sValue;

				eHWInfoAct	:= HWInfoActSetIPAddr;

				IF p_eHWInfoStat = HWInfoActSetIPAddr AND p_eHWInfoStatus = Done THEN
					eHWInfoAct	:= HWInfoActIdle;

					bUpdateP1021Network	:= TRUE;

					usiSaveIPAddrStep	:= 0;

					tyP1021McSetGen.tyGen.tyStringIPAddr.bRtCompl	:= FALSE;

				ELSIF p_eHWInfoStatus = Error THEN
					p_tyC0008MsgBox ACCESS ADR(tyP1021McSetGen.tyMsgBoxUpdtIPAddrErr);

					IF tyP1021McSetGen.tyMsgBoxUpdtIPAddrErr.tyBtnNo.bRtCompl = TRUE THEN
						tyP1021McSetGen.tyMsgBoxUpdtIPAddrErr.tyBtnNo.bRtCompl	:= FALSE;
						tyP1021McSetGen.tyMsgBoxUpdtIPAddrErr.tyBtnNo.bValue	:= FALSE;

						p_tyC0008MsgBox ACCESS ADR(tyP1021McSetGen.tyMsgBoxHide);

						//Recover IP Address
						tyP1021McSetGen.tyGen.tyStringIPAddr.sValue	:= p_sHWInfoIPAddr;

						usiSaveIPAddrStep	:= 0;

						tyP1021McSetGen.tyGen.tyStringIPAddr.bRtCompl	:= FALSE;

					END_IF

				END_IF

			END_IF

		ELSE

			p_tyC0008MsgBox ACCESS ADR(tyP1021McSetGen.tyMsgBoxIPAddrInvalid);

			IF tyP1021McSetGen.tyMsgBoxIPAddrInvalid.tyBtnNo.bRtCompl = TRUE THEN
				tyP1021McSetGen.tyMsgBoxIPAddrInvalid.tyBtnNo.bRtCompl	:= FALSE;
				tyP1021McSetGen.tyMsgBoxIPAddrInvalid.tyBtnNo.bValue	:= FALSE;

				p_tyC0008MsgBox ACCESS ADR(tyP1021McSetGen.tyMsgBoxHide);

				//Recover IP Address
				tyP1021McSetGen.tyGen.tyStringIPAddr.sValue	:= p_sHWInfoIPAddr;

				tyP1021McSetGen.tyGen.tyStringIPAddr.bRtCompl	:= FALSE;

			END_IF

		END_IF

	END_IF

END_ACTION
```

#### Act_OptP1021SubnetMask.st
```iecst
ACTION Act_OptP1021SubnetMask:

	IF tyP1021McSetGen.tyGen.tyStringSubnetMask.bRtCompl = TRUE THEN

		IF fIPValid(tyP1021McSetGen.tyGen.tyStringSubnetMask.sValue , ADR(a_iSubnetMaskPart1)) THEN

			IF usiSaveSubnetMaskStep = 0 THEN
				p_tyC0008MsgBox ACCESS ADR(tyP1021McSetGen.tyMsgBoxUpdtSubnetAsk);

				IF tyP1021McSetGen.tyMsgBoxUpdtSubnetAsk.tyBtnYes.bRtCompl = TRUE THEN
					tyP1021McSetGen.tyMsgBoxUpdtSubnetAsk.tyBtnYes.bRtCompl	:= FALSE;
					tyP1021McSetGen.tyMsgBoxUpdtSubnetAsk.tyBtnYes.bValue	:= FALSE;

					p_tyC0008MsgBox ACCESS ADR(tyP1021McSetGen.tyMsgBoxHide);

					usiSaveSubnetMaskStep	:= 1;

				ELSIF tyP1021McSetGen.tyMsgBoxUpdtSubnetAsk.tyBtnNo.bRtCompl = TRUE THEN
					tyP1021McSetGen.tyMsgBoxUpdtSubnetAsk.tyBtnNo.bRtCompl	:= FALSE;
					tyP1021McSetGen.tyMsgBoxUpdtSubnetAsk.tyBtnNo.bValue	:= FALSE;

					p_tyC0008MsgBox ACCESS ADR(tyP1021McSetGen.tyMsgBoxHide);

					//Recover Subnet Mask
					tyP1021McSetGen.tyGen.tyStringSubnetMask.sValue	:= p_sHWInfoSubnetMask;

					tyP1021McSetGen.tyGen.tyStringSubnetMask.bRtCompl	:= FALSE;

				END_IF

			ELSIF usiSaveSubnetMaskStep = 1 THEN
				//Set Subnet Mask
				sSetSubnetMask	:= tyP1021McSetGen.tyGen.tyStringSubnetMask.sValue;

				eHWInfoAct	:= HWInfoActSetSubnetMask;

				IF p_eHWInfoStat = HWInfoActSetSubnetMask AND p_eHWInfoStatus = Done THEN
					eHWInfoAct	:= HWInfoActIdle;

					bUpdateP1021Network	:= TRUE;

					usiSaveSubnetMaskStep	:= 0;

					tyP1021McSetGen.tyGen.tyStringSubnetMask.bRtCompl	:= FALSE;

				ELSIF p_eHWInfoStatus = Error THEN
					p_tyC0008MsgBox ACCESS ADR(tyP1021McSetGen.tyMsgBoxUpdtSubnetErr);

					IF tyP1021McSetGen.tyMsgBoxUpdtSubnetErr.tyBtnNo.bRtCompl = TRUE THEN
						tyP1021McSetGen.tyMsgBoxUpdtSubnetErr.tyBtnNo.bRtCompl	:= FALSE;
						tyP1021McSetGen.tyMsgBoxUpdtSubnetErr.tyBtnNo.bValue	:= FALSE;

						p_tyC0008MsgBox ACCESS ADR(tyP1021McSetGen.tyMsgBoxHide);

						//Recover Subnet Mask
						tyP1021McSetGen.tyGen.tyStringSubnetMask.sValue	:= p_sHWInfoSubnetMask;

						usiSaveSubnetMaskStep	:= 0;

						tyP1021McSetGen.tyGen.tyStringSubnetMask.bRtCompl	:= FALSE;

					END_IF

				END_IF

			END_IF

		ELSE

			p_tyC0008MsgBox ACCESS ADR(tyP1021McSetGen.tyMsgBoxSubnetInvalid);

			IF tyP1021McSetGen.tyMsgBoxSubnetInvalid.tyBtnNo.bRtCompl = TRUE THEN
				tyP1021McSetGen.tyMsgBoxSubnetInvalid.tyBtnNo.bRtCompl	:= FALSE;
				tyP1021McSetGen.tyMsgBoxSubnetInvalid.tyBtnNo.bValue	:= FALSE;

				p_tyC0008MsgBox ACCESS ADR(tyP1021McSetGen.tyMsgBoxHide);

				//Recover Subnet Mask
				tyP1021McSetGen.tyGen.tyStringSubnetMask.sValue	:= p_sHWInfoSubnetMask;

				tyP1021McSetGen.tyGen.tyStringSubnetMask.bRtCompl	:= FALSE;

			END_IF

		END_IF

	END_IF

END_ACTION
```

#### Act_OptP1021DHCPSetting.st
```iecst
ACTION Act_OptP1021DHCPSetting:

	IF p_tyMcParamCurr.eNetworkMod = IPFromDHCPServer  THEN
		fUIInRtStatOff(ADR(tyP1021McSetGen.tyGen.tyStringIPAddr.uiMaskRtStat));
		fUIInRtStatOff(ADR(tyP1021McSetGen.tyGen.tyStringSubnetMask.uiMaskRtStat));
	ELSE
		fUIInRtStatHide(ADR(tyP1021McSetGen.tyGen.tyStringIPAddr.uiMaskRtStat));
		fUIInRtStatHide(ADR(tyP1021McSetGen.tyGen.tyStringSubnetMask.uiMaskRtStat));
	END_IF

	//Trigger Save Condition
	IF tyP1021McSetGen.tyGen.tyDrpDnNetworkMod.bRtCompl THEN

		bSaveNetworkPriority := TRUE;

		usiNetworkModeNew := tyP1021McSetGen.tyGen.tyDrpDnNetworkMod.usiValueIdx;

		fUIInRtStatHide(ADR(tyCommon.tySet.tyBtnSave.uiMaskRtStat));

		tyP1021McSetGen.tyGen.tyDrpDnNetworkMod.bRtCompl := FALSE;

		IF usiNetworkModeOld<>usiNetworkModeNew THEN
			IF tyP1021McSetGen.tyGen.tyDrpDnNetworkMod.usiValueIdx = DINT_TO_USINT(SetIPManually) THEN

				tyP1021McSetGen.tyNetwork.tyStringIPAddr.sValue		:= p_sHWInfoIPAddr;
				tyP1021McSetGen.tyNetwork.tyStringSubnetMask.sValue	:= p_sHWInfoSubnetMask;
				fUIInRtStatOff(ADR(tyP1021McSetGen.tyNetwork.tyLyr.uiRtStat));

			END_IF
		END_IF

	END_IF

	// If Change from DHCP to Manual, Pop Up Detail to fill in
	IF tyP1021McSetGen.tyNetwork.tyLyr.uiRtStat.0 = FALSE THEN
		//IP Check
		IF tyP1021McSetGen.tyNetwork.tyStringIPAddr.bRtCompl = TRUE THEN
			IF fIPValid(tyP1021McSetGen.tyNetwork.tyStringIPAddr.sValue , ADR(a_iIPPart1)) THEN

				tyP1021McSetGen.tyNetwork.tyStringIPAddr.bRtCompl	:= FALSE;
			ELSE
				p_tyC0008MsgBox ACCESS ADR(tyP1021McSetGen.tyMsgBoxIPAddrInvalidEdit);

				IF tyP1021McSetGen.tyMsgBoxIPAddrInvalidEdit.tyBtnNo.bRtCompl = TRUE THEN
					tyP1021McSetGen.tyMsgBoxIPAddrInvalidEdit.tyBtnNo.bRtCompl	:= FALSE;
					tyP1021McSetGen.tyMsgBoxIPAddrInvalidEdit.tyBtnNo.bValue	:= FALSE;

					p_tyC0008MsgBox ACCESS ADR(tyP1021McSetGen.tyMsgBoxHide);

					//Recover IP Address
					tyP1021McSetGen.tyNetwork.tyStringIPAddr.sValue	:= p_sHWInfoIPAddr;
					tyP1021McSetGen.tyNetwork.tyStringIPAddr.bRtCompl	:= FALSE;
				END_IF
			END_IF
		END_IF

		//Subnet Check
		IF tyP1021McSetGen.tyNetwork.tyStringSubnetMask.bRtCompl = TRUE THEN
			IF fIPValid(tyP1021McSetGen.tyNetwork.tyStringSubnetMask.sValue , ADR(a_iSubnetMaskPart1)) THEN

				tyP1021McSetGen.tyNetwork.tyStringSubnetMask.bRtCompl	:= FALSE;
			ELSE
				p_tyC0008MsgBox ACCESS ADR(tyP1021McSetGen.tyMsgBoxSubnetInvalidEdit);

				IF tyP1021McSetGen.tyMsgBoxSubnetInvalidEdit.tyBtnNo.bRtCompl = TRUE THEN
					tyP1021McSetGen.tyMsgBoxSubnetInvalidEdit.tyBtnNo.bRtCompl	:= FALSE;
					tyP1021McSetGen.tyMsgBoxSubnetInvalidEdit.tyBtnNo.bValue	:= FALSE;

					p_tyC0008MsgBox ACCESS ADR(tyP1021McSetGen.tyMsgBoxHide);
					//Recover IP Address
					tyP1021McSetGen.tyNetwork.tyStringSubnetMask.sValue	:= p_sHWInfoSubnetMask;
					tyP1021McSetGen.tyNetwork.tyStringSubnetMask.bRtCompl	:= FALSE;

				END_IF
			END_IF
		END_IF

		IF tyP1021McSetGen.tyNetwork.tyBtnSave.bRtCompl = TRUE THEN

			tyP1021McSetGen.tyNetwork.tyBtnSave.bRtCompl	:= FALSE;
			tyP1021McSetGen.tyNetwork.tyBtnSave.bValue		:= FALSE;

			tyP1021McSetGen.tyGen.tyStringIPAddr.sValue 	:= tyP1021McSetGen.tyNetwork.tyStringIPAddr.sValue;
			tyP1021McSetGen.tyGen.tyStringSubnetMask.sValue := tyP1021McSetGen.tyNetwork.tyStringSubnetMask.sValue;

			fUIInRtStatHide(ADR(tyP1021McSetGen.tyNetwork.tyLyr.uiRtStat));

		ELSIF tyP1021McSetGen.tyNetwork.tyBtnCancel.bRtCompl = TRUE THEN
			tyP1021McSetGen.tyNetwork.tyBtnCancel.bRtCompl	:= FALSE;
			tyP1021McSetGen.tyNetwork.tyBtnCancel.bValue	:= FALSE;

			fUIInRtStatHide(ADR(tyP1021McSetGen.tyNetwork.tyLyr.uiRtStat));

		END_IF

	END_IF

	//Once click save, change config
	IF tyCommon.tySet.tyBtnSave.bRtCompl = TRUE AND bSaveNetworkPriority AND NOT bNetworkConfigChanged THEN

		IF usiNetworkModeOld<>usiNetworkModeNew THEN

			IF usiChgNetworkConfigStep = 0 THEN

				IF usiNetworkModeNew = DINT_TO_USINT(IPFromDHCPServer) THEN
					tyP1021McSetGen.tyMsgBoxChgNetworkAsk.tyTxtMsg.usiValueIdx := 189;
				ELSE
					tyP1021McSetGen.tyMsgBoxChgNetworkAsk.tyTxtMsg.usiValueIdx := 190;
				END_IF

				p_tyC0008MsgBox ACCESS ADR(tyP1021McSetGen.tyMsgBoxChgNetworkAsk);

				IF tyP1021McSetGen.tyMsgBoxChgNetworkAsk.tyBtnYes.bRtCompl = TRUE THEN
					tyP1021McSetGen.tyMsgBoxChgNetworkAsk.tyBtnYes.bRtCompl	:= FALSE;
					tyP1021McSetGen.tyMsgBoxChgNetworkAsk.tyBtnYes.bValue	:= FALSE;

					p_tyC0008MsgBox ACCESS ADR(tyP1021McSetGen.tyMsgBoxHide);

					usiChgNetworkConfigStep	:= 1;

				ELSIF tyP1021McSetGen.tyMsgBoxChgNetworkAsk.tyBtnNo.bRtCompl = TRUE THEN
					tyP1021McSetGen.tyMsgBoxChgNetworkAsk.tyBtnNo.bRtCompl	:= FALSE;
					tyP1021McSetGen.tyMsgBoxChgNetworkAsk.tyBtnNo.bValue	:= FALSE;

					tyP1021McSetGen.tyGen.tyStringIPAddr.sValue		:= p_sHWInfoIPAddr;
					tyP1021McSetGen.tyGen.tyStringSubnetMask.sValue := p_sHWInfoSubnetMask;

					//Recover Old Dropdown Value
					tyP1021McSetGen.tyGen.tyDrpDnNetworkMod.usiValueIdx	:= usiNetworkModeOld;

					//Reset Save Priority
					bSaveNetworkPriority := FALSE;

					//Reset Network Step
					usiChgNetworkConfigStep	:= 0;

					p_tyC0008MsgBox ACCESS ADR(tyP1021McSetGen.tyMsgBoxHide);

				END_IF

			ELSIF usiChgNetworkConfigStep = 1 THEN

				IF usiNetworkModeNew = DINT_TO_USINT(IPFromDHCPServer) THEN
					usiNetworkModeSelected := DINT_TO_USINT(IPFromDHCPServer);
				ELSE
					usiNetworkModeSelected := DINT_TO_USINT(SetIPManually);
				END_IF

				eHWInfoAct	:= HWInfoActSetEthConfigMode;

				IF p_eHWInfoStat = HWInfoActSetEthConfigMode AND p_eHWInfoStatus = Done THEN
					eHWInfoAct	:= HWInfoActIdle;

					usiChgNetworkConfigStep	:= 2;

				ELSIF p_eHWInfoStatus = Error THEN
					p_tyC0008MsgBox ACCESS ADR(tyP1021McSetGen.tyMsgBoxSetDHCPError);

					IF tyP1021McSetGen.tyMsgBoxSetDHCPError.tyBtnNo.bRtCompl = TRUE THEN
						tyP1021McSetGen.tyMsgBoxSetDHCPError.tyBtnNo.bRtCompl	:= FALSE;
						tyP1021McSetGen.tyMsgBoxSetDHCPError.tyBtnNo.bValue	:= FALSE;

						p_tyC0008MsgBox ACCESS ADR(tyP1021McSetGen.tyMsgBoxHide);

						//Recover Old Dropdown Value
						tyP1021McSetGen.tyGen.tyDrpDnNetworkMod.usiValueIdx	:= usiNetworkModeOld;

						//Reset Network Step
						usiChgNetworkConfigStep	:= 0;

						//Reset Save Priority
						bSaveNetworkPriority := FALSE;

					END_IF
				END_IF

			ELSIF usiChgNetworkConfigStep = 2 THEN

				IF p_eHWInfoStat = HWInfoActIdle THEN

					usiChgNetworkConfigStep := 0;
					bNetworkConfigChanged := TRUE;

				END_IF

			END_IF

		ELSE
			//Reset Save Priority
			bSaveNetworkPriority := FALSE;
		END_IF

	END_IF

	//Refresh/Set IP Address and Subnet Mask
	IF bNetworkConfigChanged THEN

		IF usiRefreshDetailStep = 0 THEN
			IF usiNetworkModeNew = DINT_TO_USINT(IPFromDHCPServer) THEN

				eHWInfoAct	:= HWInfoActGetIPAddr;

				IF p_eHWInfoStat = HWInfoActGetIPAddr AND p_eHWInfoStatus = Done THEN
					eHWInfoAct	:= HWInfoActIdle;

					usiRefreshDetailStep	:= 1;

					//Refresh IP value
					tyP1021McSetGen.tyGen.tyStringIPAddr.sValue := p_sHWInfoIPAddr;

				ELSIF p_eHWInfoStatus = Error THEN
					p_tyC0008MsgBox ACCESS ADR(tyP1021McSetGen.tyMsgBoxGetIPAddrErr);

					IF tyP1021McSetGen.tyMsgBoxGetIPAddrErr.tyBtnNo.bRtCompl = TRUE THEN
						tyP1021McSetGen.tyMsgBoxGetIPAddrErr.tyBtnNo.bRtCompl	:= FALSE;
						tyP1021McSetGen.tyMsgBoxGetIPAddrErr.tyBtnNo.bValue	:= FALSE;

						p_tyC0008MsgBox ACCESS ADR(tyP1021McSetGen.tyMsgBoxHide);

						//Reset Save Priority
						bSaveNetworkPriority := FALSE;

						//Reset Refresh Step
						usiRefreshDetailStep	:= 0;

						bNetworkConfigChanged	:= FALSE;

					END_IF
				END_IF

			ELSE
				eHWInfoAct	:= HWInfoActSetIPAddr;

				sSetIPAddr	:= tyP1021McSetGen.tyGen.tyStringIPAddr.sValue;

				IF p_eHWInfoStat = HWInfoActSetIPAddr AND p_eHWInfoStatus = Done THEN
					eHWInfoAct	:= HWInfoActIdle;

					usiRefreshDetailStep	:= 1;

				ELSIF p_eHWInfoStatus = Error THEN
					p_tyC0008MsgBox ACCESS ADR(tyP1021McSetGen.tyMsgBoxUpdtIPAddrErr);

					IF tyP1021McSetGen.tyMsgBoxUpdtIPAddrErr.tyBtnNo.bRtCompl = TRUE THEN
						tyP1021McSetGen.tyMsgBoxUpdtIPAddrErr.tyBtnNo.bRtCompl	:= FALSE;
						tyP1021McSetGen.tyMsgBoxUpdtIPAddrErr.tyBtnNo.bValue	:= FALSE;

						p_tyC0008MsgBox ACCESS ADR(tyP1021McSetGen.tyMsgBoxHide);

						tyP1021McSetGen.tyGen.tyStringIPAddr.sValue := p_sHWInfoIPAddr;

						//Reset Save Priority
						bSaveNetworkPriority := FALSE;

						//Reset Refresh Step
						usiRefreshDetailStep	:= 0;

						bNetworkConfigChanged	:= FALSE;

					END_IF
				END_IF
			END_IF

		ELSIF usiRefreshDetailStep = 1 THEN

			IF p_eHWInfoStat = HWInfoActIdle THEN
				usiRefreshDetailStep := 2;
			END_IF

		ELSIF usiRefreshDetailStep = 2 THEN
			IF usiNetworkModeNew = DINT_TO_USINT(IPFromDHCPServer) THEN

				eHWInfoAct	:= HWInfoActGetSubnetMask;

				IF p_eHWInfoStat = HWInfoActGetSubnetMask AND p_eHWInfoStatus = Done THEN
					eHWInfoAct	:= HWInfoActIdle;

					//Reset Save Priority
					bSaveNetworkPriority := FALSE;

					//Reset Refresh Step
					usiRefreshDetailStep	:= 0;

					//Refresh subnet value
					tyP1021McSetGen.tyGen.tyStringSubnetMask.sValue := p_sHWInfoSubnetMask;

					bNetworkConfigChanged	:= FALSE;

				ELSIF p_eHWInfoStatus = Error THEN
					p_tyC0008MsgBox ACCESS ADR(tyP1021McSetGen.tyMsgBoxGetSubnetErr);

					IF tyP1021McSetGen.tyMsgBoxGetSubnetErr.tyBtnNo.bRtCompl = TRUE THEN
						tyP1021McSetGen.tyMsgBoxGetSubnetErr.tyBtnNo.bRtCompl	:= FALSE;
						tyP1021McSetGen.tyMsgBoxGetSubnetErr.tyBtnNo.bValue	:= FALSE;

						p_tyC0008MsgBox ACCESS ADR(tyP1021McSetGen.tyMsgBoxHide);

						//Reset Save Priority
						bSaveNetworkPriority := FALSE;

						//Reset Refresh Step
						usiRefreshDetailStep	:= 0;

						bNetworkConfigChanged	:= FALSE;

					END_IF
				END_IF

			ELSE
				eHWInfoAct	:= HWInfoActSetSubnetMask;

				sSetSubnetMask	:= tyP1021McSetGen.tyGen.tyStringSubnetMask.sValue;

				IF p_eHWInfoStat = HWInfoActSetSubnetMask AND p_eHWInfoStatus = Done THEN
					eHWInfoAct	:= HWInfoActIdle;

					//Reset Save Priority
					bSaveNetworkPriority := FALSE;

					//Reset Refresh Step
					usiRefreshDetailStep	:= 0;

					bNetworkConfigChanged	:= FALSE;

				ELSIF p_eHWInfoStatus = Error THEN
					p_tyC0008MsgBox ACCESS ADR(tyP1021McSetGen.tyMsgBoxUpdtSubnetErr);

					IF tyP1021McSetGen.tyMsgBoxUpdtSubnetErr.tyBtnNo.bRtCompl = TRUE THEN
						tyP1021McSetGen.tyMsgBoxUpdtSubnetErr.tyBtnNo.bRtCompl	:= FALSE;
						tyP1021McSetGen.tyMsgBoxUpdtSubnetErr.tyBtnNo.bValue	:= FALSE;

						p_tyC0008MsgBox ACCESS ADR(tyP1021McSetGen.tyMsgBoxHide);

						tyP1021McSetGen.tyGen.tyStringSubnetMask.sValue := p_sHWInfoSubnetMask;

						//Reset Save Priority
						bSaveNetworkPriority := FALSE;

						//Reset Refresh Step
						usiRefreshDetailStep	:= 0;

						bNetworkConfigChanged	:= FALSE;

					END_IF
				END_IF
			END_IF

		END_IF
	END_IF

END_ACTION
```

#### Act_EntP1022Disp.st
```iecst
ACTION Act_EntP1022Disp:

	//Access Address
			//new for Hermes 1.3
	IF p_tyNtParamCurr.bLFPrep OR p_tyNtParamCurr.bLCSLFPrep OR p_tyNtParamCurr.bLCSReqRcpPrep OR p_tyNtParamCurr.bLCSManageRcpPrep OR p_tyNtParamCurr.bLCSLiveDatPrep
		OR p_tyNtParamCurr.bLFUsrSetPrep OR p_tyNtParamCurr.bLFUsrSetPrep OR  p_tyNtParamCurr.bUSWidthChkPrep OR p_tyNtParamCurr.bDSWidthChkPrep THEN
		bNaviLyr1 := TRUE;
	ELSE
		bNaviLyr1 := FALSE;
	END_IF

	IF (p_tyNtParamCurr.bHermesSvyPrep AND p_tyMcParamCurr.bHermesSvyEn)  THEN
		bNaviLyr2 := TRUE;
	ELSE
		bNaviLyr2 := FALSE;
	END_IF

	IF bNaviLyr1 AND NOT bNaviLyr2 THEN
		p_tyC0004Navi ACCESS ADR(tyP1022McSetVComm.tyNaviLyr1);
		fUIInRtStatOff(ADR(tyP1022McSetVComm.tyVComSel.tyLyr.uiRtStat)); //show
		fUIInRtStatHide(ADR(tyP1022McSetVComm.tyVComSvy.tyLyr.uiRtStat));
		fUIInRtStatOff(ADR(tyP1022McSetVComm.tyLF.tyLyr.uiRtStat)); //show

	ELSIF NOT bNaviLyr1 AND bNaviLyr2 THEN
		p_tyC0004Navi ACCESS ADR(tyP1022McSetVComm.tyNaviLyr2);
		fUIInRtStatHide(ADR(tyP1022McSetVComm.tyVComSel.tyLyr.uiRtStat)); //show
		fUIInRtStatOff(ADR(tyP1022McSetVComm.tyVComSvy.tyLyr.uiRtStat));
		fUIInRtStatHide(ADR(tyP1022McSetVComm.tyLF.tyLyr.uiRtStat)); //show

	ELSIF bNaviLyr1 AND bNaviLyr2 THEN
		p_tyC0004Navi ACCESS ADR(tyP1022McSetVComm.tyNaviLyr3);
		fUIInRtStatOff(ADR(tyP1022McSetVComm.tyVComSel.tyLyr.uiRtStat)); //show
		fUIInRtStatHide(ADR(tyP1022McSetVComm.tyVComSvy.tyLyr.uiRtStat));
		fUIInRtStatOff(ADR(tyP1022McSetVComm.tyLF.tyLyr.uiRtStat)); //show
	END_IF

//	p_tyC0004Navi ACCESS ADR(tyP1022McSetVComm.tyNaviBack);

	p_tyC0005Main ACCESS ADR(tyCommon.tyMain);

	p_tyC0006Set ACCESS ADR(tyCommon.tySet);

	p_tyC0007Notif ACCESS ADR(tyCommon.tyNotif);

	p_tyC0008MsgBox ACCESS ADR(tyP1022McSetVComm.tyMsgBoxHide);

	p_tyC0009Info ACCESS ADR(tyCommon.tyInfo);

	p_tyC0011Loading ACCESS ADR(tyCommon.tyLoading);

	p_tyP1022McSetVCommSel ACCESS ADR(tyP1022McSetVComm.tyVComSel);
	p_tyP1022McSetVCommLF ACCESS ADR(tyP1022McSetVComm.tyLF);
	p_tyP1022McSetVCommSvy ACCESS ADR(tyP1022McSetVComm.tyVComSvy); //new for Hermes 1.3
																(*ADD for 2023-0061E01*)
	IF p_tyNtParamCurr.bHermesSvyFirstMcInTheLine = FALSE AND p_tyNtParamCurr.bHermesSvyQueryBoardInfo = FALSE THEN
		fUIInRtStatHide(ADR(tyP1022McSetVComm.tyVComSvy.tyBtnQueryWorkOrderInfo.uiRtStat));
	END_IF

	//Backup Param
	tyP1022McSetVComm.tyVComSelBkUp	:= tyP1022McSetVComm.tyVComSel;
	tyP1022McSetVComm.tyLFBkUp		:= tyP1022McSetVComm.tyLF;
	tyP1022McSetVComm.tyVComSvyBkUp	:= tyP1022McSetVComm.tyVComSvy; //new for Hermes 1.3

END_ACTION
```

#### Act_ExitP1022.st
```iecst
ACTION Act_ExitP1022:

	IF tyCommon.tySet.tyBtnSave.uiMaskRtStat.0 = FALSE THEN
		usiChgPage	:= 1;

	ELSE

		p_tyC0008MsgBox ACCESS ADR(tyP1022McSetVComm.tyMsgBoxExitAsk);

		IF tyP1022McSetVComm.tyMsgBoxExitAsk.tyBtnYes.bRtCompl = TRUE THEN
			tyP1022McSetVComm.tyMsgBoxExitAsk.tyBtnYes.bRtCompl	:= FALSE;
			tyP1022McSetVComm.tyMsgBoxExitAsk.tyBtnYes.bValue	:= FALSE;

			p_tyC0008MsgBox ACCESS ADR(tyP1022McSetVComm.tyMsgBoxHide);

			//Restore Param
			tyP1022McSetVComm.tyVComSel	:= tyP1022McSetVComm.tyVComSelBkUp;
			tyP1022McSetVComm.tyLF		:= tyP1022McSetVComm.tyLFBkUp;
			tyP1022McSetVComm.tyVComSvy	:= tyP1022McSetVComm.tyVComSvyBkUp; //new for Hermes 1.3

			fUIInRtStatOff(ADR(tyCommon.tySet.tyBtnSave.uiMaskRtStat));

			usiChgPage	:= 1;

		ELSIF tyP1022McSetVComm.tyMsgBoxExitAsk.tyBtnNo.bRtCompl = TRUE THEN
			tyP1022McSetVComm.tyMsgBoxExitAsk.tyBtnNo.bRtCompl	:= FALSE;
			tyP1022McSetVComm.tyMsgBoxExitAsk.tyBtnNo.bValue	:= FALSE;

			p_tyC0008MsgBox ACCESS ADR(tyP1022McSetVComm.tyMsgBoxHide);

			eChgPage	:= eCurrPage;
			usiChgPage	:= 0;

		END_IF

	END_IF

END_ACTION
```

#### Act_OptP1022Navi.st
```iecst
ACTION Act_OptP1022Navi:

//	//tyP1022McSetVComm.tyNaviBack.tyBtnBack.bRtLk	:= tyCommon.tySet.tyBtnSave.bRtCompl;
//
//	IF tyP1022McSetVComm.tyNaviBack.tyBtnBack.bRtCompl = TRUE THEN
//		eChgPage	:= UIP1020McSetNavi;
//
//		tyP1022McSetVComm.tyNaviBack.tyBtnBack.bRtCompl	:= FALSE;
//
//	END_IF

	tyP1022McSetVComm.tyNaviBack.tyBtnBack.bRtLk	:= tyCommon.tySet.tyBtnSave.bRtCompl;

	IF tyP1022McSetVComm.tyNaviLyr1.tyBtnBack.bRtCompl OR tyP1022McSetVComm.tyNaviLyr2.tyBtnBack.bRtCompl OR
		tyP1022McSetVComm.tyNaviLyr3.tyBtnBack.bRtCompl OR tyP1022McSetVComm.tyNaviLyr4.tyBtnBack.bRtCompl THEN
		tyP1022McSetVComm.tyNaviLyr1.tyBtnBack.bRtCompl	:= FALSE;
		tyP1022McSetVComm.tyNaviLyr2.tyBtnBack.bRtCompl	:= FALSE;
		tyP1022McSetVComm.tyNaviLyr3.tyBtnBack.bRtCompl	:= FALSE;
		tyP1022McSetVComm.tyNaviLyr4.tyBtnBack.bRtCompl	:= FALSE;

		eChgPage	:= UIP1020McSetNavi;

	ELSIF tyP1022McSetVComm.tyNaviLyr3.tyBtnLeft.bRtCompl = TRUE OR tyP1022McSetVComm.tyNaviLyr3.tyBtnRgt.bRtCompl = TRUE THEN
		tyP1022McSetVComm.tyNaviLyr3.tyBtnLeft.bRtCompl	:= FALSE;
		tyP1022McSetVComm.tyNaviLyr3.tyBtnRgt.bRtCompl	:= FALSE;

		p_tyC0004Navi ACCESS ADR(tyP1022McSetVComm.tyNaviLyr4);

		fUIInRtStatHide(ADR(tyP1022McSetVComm.tyVComSel.tyLyr.uiRtStat));
		fUIInRtStatOff(ADR(tyP1022McSetVComm.tyVComSvy.tyLyr.uiRtStat)); //new for Hermes 1.3
		fUIInRtStatHide(ADR(tyP1022McSetVComm.tyLF.tyLyr.uiRtStat));

	ELSIF tyP1022McSetVComm.tyNaviLyr4.tyBtnLeft.bRtCompl = TRUE OR tyP1022McSetVComm.tyNaviLyr4.tyBtnRgt.bRtCompl = TRUE THEN
		tyP1022McSetVComm.tyNaviLyr4.tyBtnLeft.bRtCompl	:= FALSE;
		tyP1022McSetVComm.tyNaviLyr4.tyBtnRgt.bRtCompl	:= FALSE;

		p_tyC0004Navi ACCESS ADR(tyP1022McSetVComm.tyNaviLyr3);

		fUIInRtStatOff(ADR(tyP1022McSetVComm.tyVComSel.tyLyr.uiRtStat));
		fUIInRtStatHide(ADR(tyP1022McSetVComm.tyVComSvy.tyLyr.uiRtStat));  //new for Hermes 1.3
		fUIInRtStatOff(ADR(tyP1022McSetVComm.tyLF.tyLyr.uiRtStat));
	END_IF

END_ACTION
```

#### Act_OptP1022Save.st
```iecst
ACTION Act_OptP1022Save:

	IF tyP1022McSetVComm.tyVComSel.tyBtnLF.bRtCompl 			OR tyP1022McSetVComm.tyVComSel.tyBtnLCSLF.bRtCompl
		OR tyP1022McSetVComm.tyVComSel.tyBtnLCSReqRcp.bRtCompl	OR tyP1022McSetVComm.tyVComSel.tyBtnLCSManageRcp.bRtCompl
		OR tyP1022McSetVComm.tyVComSel.tyBtnLCSLiveDat.bRtCompl	OR tyP1022McSetVComm.tyLF.tyBtnSectionLdr.bRtCompl
		OR tyP1022McSetVComm.tyLF.tyBtnUSWidthChkEn.bRtCompl	OR tyP1022McSetVComm.tyLF.tyBtnDSWidthChkEn.bRtCompl
		OR tyP1022McSetVComm.tyLF.tyBtnLeaderMc.bRtCompl 		OR tyP1022McSetVComm.tyLF.tyBtnSeqStayActive.bRtCompl
		OR tyP1022McSetVComm.tyVComSvy.tyBtnConfiguration.bRtCompl //new for Hermes 1.3
		OR tyP1022McSetVComm.tyVComSvy.tyBtnCheckAliveResponse.bRtCompl OR tyP1022McSetVComm.tyVComSvy.tyBtnBoardTracking.bRtCompl //new for Hermes 1.3
		OR tyP1022McSetVComm.tyVComSvy.tyBtnQueryWorkOrderInfo.bRtCompl OR tyP1022McSetVComm.tyVComSvy.tyBtnSendWorkOrderInfo.bRtCompl //new for Hermes 1.3
		OR tyP1022McSetVComm.tyVComSvy.tyNumSndAliveTm.bRtCompl         OR tyP1022McSetVComm.tyVComSvy.tyNumSvySystemPort.bRtCompl //new for Hermes 1.3
		OR tyP1022McSetVComm.tyLF.tyBtnDBAOnWOAlign.bRtCompl	THEN

		fUIInRtStatHide(ADR(tyCommon.tySet.tyBtnSave.uiMaskRtStat));

		IF (NOT p_tyNtParamCurr.bLFUsrSetPrep AND NOT p_tyNtParamCurr.bLeaderMc) OR (p_tyNtParamCurr.bLFUsrSetPrep AND NOT tyP1022McSetVComm.tyLF.tyBtnLeaderMc.bValue) THEN
			IF tyP1022McSetVComm.tyVComSel.tyBtnLF.bRtCompl AND tyP1022McSetVComm.tyVComSel.tyBtnLF.bValue THEN
				tyP1022McSetVComm.tyVComSel.tyBtnLCSLF.bValue	:= FALSE;

			ELSIF tyP1022McSetVComm.tyVComSel.tyBtnLCSLF.bRtCompl AND tyP1022McSetVComm.tyVComSel.tyBtnLCSLF.bValue THEN
				tyP1022McSetVComm.tyVComSel.tyBtnLF.bValue		:= FALSE;

			END_IF

			IF tyP1022McSetVComm.tyVComSel.tyBtnLF.bValue = TRUE AND tyP1022McSetVComm.tyVComSel.tyBtnLCSLF.bValue = TRUE THEN
				tyP1022McSetVComm.tyVComSel.tyBtnLF.bValue		:= FALSE;
				tyP1022McSetVComm.tyVComSel.tyBtnLCSLF.bValue	:= FALSE;
			END_IF
		END_IF

		tyP1022McSetVComm.tyVComSel.tyBtnLF.bRtCompl					:= FALSE;
		tyP1022McSetVComm.tyVComSel.tyBtnLCSLF.bRtCompl					:= FALSE;
		tyP1022McSetVComm.tyVComSel.tyBtnLCSReqRcp.bRtCompl				:= FALSE;
		tyP1022McSetVComm.tyVComSel.tyBtnLCSManageRcp.bRtCompl			:= FALSE;
		tyP1022McSetVComm.tyVComSel.tyBtnLCSLiveDat.bRtCompl			:= FALSE;

		tyP1022McSetVComm.tyLF.tyBtnLeaderMc.bRtCompl					:= FALSE;
		tyP1022McSetVComm.tyLF.tyBtnSectionLdr.bRtCompl					:= FALSE;
		tyP1022McSetVComm.tyLF.tyBtnUSWidthChkEn.bRtCompl				:= FALSE;
		tyP1022McSetVComm.tyLF.tyBtnDSWidthChkEn.bRtCompl				:= FALSE;
		tyP1022McSetVComm.tyLF.tyBtnSeqStayActive.bRtCompl				:= FALSE;
		tyP1022McSetVComm.tyLF.tyBtnDBAOnWOAlign.bRtCompl		:= FALSE;

		//new for Hermes 1.3
		tyP1022McSetVComm.tyVComSvy.tyBtnConfiguration.bRtCompl			:= FALSE;
		tyP1022McSetVComm.tyVComSvy.tyBtnCheckAliveResponse.bRtCompl	:= FALSE;
		tyP1022McSetVComm.tyVComSvy.tyBtnBoardTracking.bRtCompl			:= FALSE;
		tyP1022McSetVComm.tyVComSvy.tyBtnQueryWorkOrderInfo.bRtCompl	:= FALSE;
		tyP1022McSetVComm.tyVComSvy.tyBtnSendWorkOrderInfo.bRtCompl		:= FALSE;
		tyP1022McSetVComm.tyVComSvy.tyNumSndAliveTm.bRtCompl			:= FALSE;
		tyP1022McSetVComm.tyVComSvy.tyNumSvySystemPort.bRtCompl			:= FALSE;

	END_IF

	IF tyCommon.tySet.tyBtnSave.bRtCompl = TRUE THEN

		tyMcParamWr.bLFEn			:=  tyP1022McSetVComm.tyVComSel.tyBtnLF.bValue;
		tyMcParamWr.bLCSLFEn		:=  tyP1022McSetVComm.tyVComSel.tyBtnLCSLF.bValue;
		tyMcParamWr.bLCSReqRcpEn	:=  tyP1022McSetVComm.tyVComSel.tyBtnLCSReqRcp.bValue;
		tyMcParamWr.bLCSManageRcpEn	:=  tyP1022McSetVComm.tyVComSel.tyBtnLCSManageRcp.bValue;
		tyMcParamWr.bLCSLiveDatEn	:=  tyP1022McSetVComm.tyVComSel.tyBtnLCSLiveDat.bValue;

		tyMcParamWr.bLFLeaderMc		:=	tyP1022McSetVComm.tyLF.tyBtnLeaderMc.bValue;
		tyMcParamWr.bSectionLeader	:=	tyP1022McSetVComm.tyLF.tyBtnSectionLdr.bValue;
		tyMcParamWr.bUSWidthChkEn	:= 	tyP1022McSetVComm.tyLF.tyBtnUSWidthChkEn.bValue;
		tyMcParamWr.bDSWidthChkEn	:= 	tyP1022McSetVComm.tyLF.tyBtnDSWidthChkEn.bValue;
		tyMcParamWr.bLFSeqStayActive	:= 	tyP1022McSetVComm.tyLF.tyBtnSeqStayActive.bValue;
		tyMcParamWr.bDBAOnWOAlign		:=  tyP1022McSetVComm.tyLF.tyBtnDBAOnWOAlign.bValue;

		//new for Hermes 1.3
		tyHermesSvyParamWr.bFeatureConfiguration	    	:=	tyP1022McSetVComm.tyVComSvy.tyBtnConfiguration.bValue;
		tyHermesSvyParamWr.bFeatureCheckAliveResponse		:=	tyP1022McSetVComm.tyVComSvy.tyBtnCheckAliveResponse.bValue;
		tyHermesSvyParamWr.bFeatureBoardTracking	    	:=	tyP1022McSetVComm.tyVComSvy.tyBtnBoardTracking.bValue;
		tyHermesSvyParamWr.bFeatureQueryWorkOrderInfo		:=	tyP1022McSetVComm.tyVComSvy.tyBtnQueryWorkOrderInfo.bValue;
		tyHermesSvyParamWr.bFeatureSendWorkOrderInfo		:=	tyP1022McSetVComm.tyVComSvy.tyBtnSendWorkOrderInfo.bValue;
		tyHermesSvyParamWr.tSndAlive		                :=	DINT_TO_TIME(tyP1022McSetVComm.tyVComSvy.tyNumSndAliveTm.diValue);
		tyHermesSvyParamWr.uiSvySvstemPort		            :=	DINT_TO_UINT(tyP1022McSetVComm.tyVComSvy.tyNumSvySystemPort.diValue);
		bSaveHMISvyConfig := TRUE;

		eMcParamAct	:= McParamActWrite;
		eHermesAct	:= HermesActWriteConfig; //new for Hermes 1.3

		IF p_eMcParamStat = McParamActWrite AND p_eMcParamStatus = Done AND p_eHermesStat = HermesActWriteConfig AND p_eHermesStatus = Done THEN  //new for Hermes 1.3
			eMcParamAct	:= McParamActIdle;
			eHermesAct	:= HermesActIdle;  //new for Hermes 1.3

			//Update BackUp Param
			tyP1022McSetVComm.tyVComSelBkUp	:= tyP1022McSetVComm.tyVComSel;
			tyP1022McSetVComm.tyLFBkUp		:= tyP1022McSetVComm.tyLF;
			tyP1022McSetVComm.tyVComSvyBkUp	:= tyP1022McSetVComm.tyVComSvy;  //new for Hermes 1.3

			tyCommon.tySet.tyBtnSave.bRtCompl	:= FALSE;
			fUIInRtStatOff(ADR(tyCommon.tySet.tyBtnSave.uiMaskRtStat));
			bSaveHMISvyConfig := FALSE;  //new for Hermes 1.3

		ELSIF p_eMcParamStatus = Error OR p_eHermesStatus = Error THEN
			p_tyC0008MsgBox ACCESS ADR(tyP1022McSetVComm.tyMsgBoxSaveErr);

			IF tyP1022McSetVComm.tyMsgBoxSaveErr.tyBtnNo.bRtCompl = TRUE THEN
				tyP1022McSetVComm.tyMsgBoxSaveErr.tyBtnNo.bRtCompl 	:= FALSE;
				tyP1022McSetVComm.tyMsgBoxSaveErr.tyBtnNo.bValue	:= FALSE;

				p_tyC0008MsgBox ACCESS ADR(tyP1022McSetVComm.tyMsgBoxHide);

				//Restore Param
				tyP1022McSetVComm.tyVComSel	:= tyP1022McSetVComm.tyVComSelBkUp;
				tyP1022McSetVComm.tyVComSvy	:= tyP1022McSetVComm.tyVComSvyBkUp;  //new for Hermes 1.3
				tyP1022McSetVComm.tyLF		:= tyP1022McSetVComm.tyLFBkUp;
				tyMcParamWr					:= p_tyMcParamCurr;
				bSaveHMISvyConfig := FALSE;  //new for Hermes 1.3

				tyCommon.tySet.tyBtnSave.bRtCompl 	:= FALSE;
				fUIInRtStatOff(ADR(tyCommon.tySet.tyBtnSave.uiMaskRtStat));

			END_IF

		END_IF

	END_IF

END_ACTION
```

#### Act_OptP1022DisLF.st
```iecst
ACTION Act_OptP1022DisLF:

	IF tyP1022McSetVComm.tyVComSel.tyBtnLF.bValue=FALSE OR (tyP1022McSetVComm.tyVComSel.tyBtnLF.bValue AND tyP1022McSetVComm.tyLF.tyBtnLeaderMc.bValue=FALSE) THEN
		IF bLFRunInBG THEN
			usiLFLeaderCtrlStep	:= 0;

			eLFLeaderAct	:= LFActIdle;

			fbLFLeaderCtrlBlinkTm(IN := FALSE);

			tyP0700LFCtrl.tyLdr.tyBitmapChgAll.usiValueIdx		:= 0;
			tyP0700LFCtrl.tyLdr.tyBitmapChgSeqAuto.usiValueIdx	:= 0;
			tyP0700LFCtrl.tyLdr.tyBitmapChgSeqMnl.usiValueIdx	:= 0;
			tyP0700LFCtrl.tyLdr.tyBitmapSyncTm.usiValueIdx		:= 0;

			tyP0700LFCtrl.tyLdr.tyBtnChgAll.bRtCompl			:= FALSE;
			tyP0700LFCtrl.tyLdr.tyBtnChgSeqAuto.bRtCompl		:= FALSE;
			tyP0700LFCtrl.tyLdr.tyBtnChgSeqMnl.bRtCompl			:= FALSE;
			tyP0700LFCtrl.tyLdr.tyBtnSyncTm.bRtCompl			:= FALSE;

			tyP0700LFCtrl.tyLdr.tyBtnChgAll.bValue				:= FALSE;
			tyP0700LFCtrl.tyLdr.tyBtnChgSeqAuto.bValue			:= FALSE;
			tyP0700LFCtrl.tyLdr.tyBtnChgSeqMnl.bValue			:= FALSE;
			tyP0700LFCtrl.tyLdr.tyBtnSyncTm.bValue				:= FALSE;

			bLFRunInBG	:= FALSE;

		END_IF
	END_IF

END_ACTION
```

#### Act_EntP1023Disp.st
```iecst
ACTION Act_EntP1023Disp:

	//Access Address
	p_tyC0004Navi ACCESS ADR(tyP1023McSetHComm.tyNaviLyr1);

	p_tyC0005Main ACCESS ADR(tyCommon.tyMain);

	p_tyC0006Set ACCESS ADR(tyCommon.tySet);

	p_tyC0007Notif ACCESS ADR(tyCommon.tyNotif);

	p_tyC0008MsgBox ACCESS ADR(tyP1023McSetHComm.tyMsgBoxHide);

	p_tyC0009Info ACCESS ADR(tyCommon.tyInfo);

	p_tyC0011Loading ACCESS ADR(tyCommon.tyLoading);

	p_tyP1023McSetHCommGen ACCESS ADR(tyP1023McSetHComm.tyGen);

	p_tyP1023McSetHCommUSSel ACCESS ADR(tyP1023McSetHComm.tyUSSel);
	p_tyP1023McSetHCommDSSel ACCESS ADR(tyP1023McSetHComm.tyDSSel);
	p_tyP1023McSetHCommUSSMEMA ACCESS ADR(tyP1023McSetHComm.tyUSSMEMA);
	p_tyP1023McSetHCommDSSMEMA ACCESS ADR(tyP1023McSetHComm.tyDSSMEMA);
	p_tyP1023McSetHCommUSHermes ACCESS ADR(tyP1023McSetHComm.tyUSHermes);
	p_tyP1023McSetHCommDSHermes ACCESS ADR(tyP1023McSetHComm.tyDSHermes);

	p_tyP1023McSetHCommUSSel2 ACCESS ADR(tyP1023McSetHComm.tyUSSel2);
	p_tyP1023McSetHCommUSSMEMA2 ACCESS ADR(tyP1023McSetHComm.tyUSSMEMA2);

	//DropDown
	tyP1023McSetHComm.tyGen.tyDrpDnUSSel.usiValueIdx 	:=0;
	tyP1023McSetHComm.tyGen.tyDrpDnDSSel.usiValueIdx 	:=0;

	tyP1023McSetHComm.tyGen.tyDrpDnUSSel.usiValueMaxIdx 	:=1;
	tyP1023McSetHComm.tyGen.tyDrpDnDSSel.usiValueMaxIdx 	:=1;

	//Display
	fUIInRtStatOff(ADR(tyP1023McSetHComm.tyUSSel.tyLyr.uiRtStat));
	fUIInRtStatHide(ADR(tyP1023McSetHComm.tyDSSel.tyLyr.uiRtStat));
	fUIInRtStatHide(ADR(tyP1023McSetHComm.tyDSSMEMA.tyLyr.uiRtStat));
	fUIInRtStatHide(ADR(tyP1023McSetHComm.tyDSHermes.tyLyr.uiRtStat));
	fUIInRtStatHide(ADR(tyP1023McSetHComm.tyUSSel2.tyLyr.uiRtStat));
	fUIInRtStatHide(ADR(tyP1023McSetHComm.tyUSSMEMA2.tyLyr.uiRtStat));

	//Backup Param
	tyP1023McSetHComm.tyUSSelBkUp		:= tyP1023McSetHComm.tyUSSel;
	tyP1023McSetHComm.tyUSSMEMABkUp		:= tyP1023McSetHComm.tyUSSMEMA;
	tyP1023McSetHComm.tyUSHermesBkUp	:= tyP1023McSetHComm.tyUSHermes;
	tyP1023McSetHComm.tyDSSelBkUp		:= tyP1023McSetHComm.tyDSSel;
	tyP1023McSetHComm.tyDSSMEMABkUp		:= tyP1023McSetHComm.tyDSSMEMA;
	tyP1023McSetHComm.tyDSHermesBkUp	:= tyP1023McSetHComm.tyDSHermes;

	//Backup Param Upstream 2
	tyP1023McSetHComm.tyUSSelBkUp2		:= tyP1023McSetHComm.tyUSSel2;
	tyP1023McSetHComm.tyUSSMEMABkUp2	:= tyP1023McSetHComm.tyUSSMEMA2;
	tyP1023McSetHComm.tyUSHermesBkUp2	:= tyP1023McSetHComm.tyUSHermes2;
END_ACTION
```

#### Act_ExitP1023.st
```iecst
ACTION Act_ExitP1023:

	IF tyCommon.tySet.tyBtnSave.uiMaskRtStat.0 = FALSE THEN
		usiChgPage	:= 1;

	ELSE

		p_tyC0008MsgBox ACCESS ADR(tyP1023McSetHComm.tyMsgBoxExitAsk);

		IF tyP1023McSetHComm.tyMsgBoxExitAsk.tyBtnYes.bRtCompl = TRUE THEN
			tyP1023McSetHComm.tyMsgBoxExitAsk.tyBtnYes.bRtCompl	:= FALSE;
			tyP1023McSetHComm.tyMsgBoxExitAsk.tyBtnYes.bValue	:= FALSE;

			p_tyC0008MsgBox ACCESS ADR(tyP1023McSetHComm.tyMsgBoxHide);

			//Restore Param
			tyP1023McSetHComm.tyUSSel		:= tyP1023McSetHComm.tyUSSelBkUp;
			tyP1023McSetHComm.tyUSSMEMA		:= tyP1023McSetHComm.tyUSSMEMABkUp;
			tyP1023McSetHComm.tyUSHermes	:= tyP1023McSetHComm.tyUSHermesBkUp;
			tyP1023McSetHComm.tyDSSel		:= tyP1023McSetHComm.tyDSSelBkUp;
			tyP1023McSetHComm.tyDSSMEMA		:= tyP1023McSetHComm.tyDSSMEMABkUp;
			tyP1023McSetHComm.tyDSHermes	:= tyP1023McSetHComm.tyDSHermesBkUp;
			tyP1023McSetHComm.tyUSSel2		:= tyP1023McSetHComm.tyUSSelBkUp2;
			tyP1023McSetHComm.tyUSSMEMA2	:= tyP1023McSetHComm.tyUSSMEMABkUp2;

			fUIInRtStatOff(ADR(tyCommon.tySet.tyBtnSave.uiMaskRtStat));

			usiChgPage	:= 1;

		ELSIF tyP1023McSetHComm.tyMsgBoxExitAsk.tyBtnNo.bRtCompl = TRUE THEN
			tyP1023McSetHComm.tyMsgBoxExitAsk.tyBtnNo.bRtCompl	:= FALSE;
			tyP1023McSetHComm.tyMsgBoxExitAsk.tyBtnNo.bValue	:= FALSE;

			p_tyC0008MsgBox ACCESS ADR(tyP1023McSetHComm.tyMsgBoxHide);

			eChgPage	:= eCurrPage;
			usiChgPage	:= 0;

		END_IF

	END_IF

END_ACTION
```

#### Act_OptP1023Navi.st
```iecst
ACTION Act_OptP1023Navi:

	IF tyP1023McSetHComm.tyNaviLyr1.tyBtnBack.bRtCompl = TRUE OR tyP1023McSetHComm.tyNaviLyr2.tyBtnBack.bRtCompl = TRUE THEN
		tyP1023McSetHComm.tyNaviLyr1.tyBtnBack.bRtCompl	:= FALSE;
		tyP1023McSetHComm.tyNaviLyr2.tyBtnBack.bRtCompl	:= FALSE;

		eChgPage	:= UIP1020McSetNavi;

	ELSIF tyP1023McSetHComm.tyNaviLyr1.tyBtnLeft.bRtCompl = TRUE OR tyP1023McSetHComm.tyNaviLyr1.tyBtnRgt.bRtCompl = TRUE THEN
		tyP1023McSetHComm.tyNaviLyr1.tyBtnLeft.bRtCompl	:= FALSE;
		tyP1023McSetHComm.tyNaviLyr1.tyBtnRgt.bRtCompl	:= FALSE;

		p_tyC0004Navi ACCESS ADR(tyP1023McSetHComm.tyNaviLyr2);

		fUIInRtStatHide(ADR(tyP1023McSetHComm.tyUSSel.tyLyr.uiRtStat));
		fUIInRtStatHide(ADR(tyP1023McSetHComm.tyUSSel2.tyLyr.uiRtStat));

		IF tyP1023McSetHComm.tyGen.tyDrpDnDSSel.usiValueIdx = 0 THEN

			p_tyP1023McSetHCommDSSel ACCESS ADR(tyP1023McSetHComm.tyDSSel);
			p_tyP1023McSetHCommDSSMEMA ACCESS ADR(tyP1023McSetHComm.tyDSSMEMA);
			p_tyP1023McSetHCommDSHermes ACCESS ADR(tyP1023McSetHComm.tyDSHermes);

			fUIInRtStatOff(ADR(tyP1023McSetHComm.tyDSSel.tyLyr.uiRtStat));
			fUIInRtStatHide(ADR(tyP1023McSetHComm.tyDSSel2.tyLyr.uiRtStat));

		ELSIF tyP1023McSetHComm.tyGen.tyDrpDnDSSel.usiValueIdx = 1 THEN

			p_tyP1023McSetHCommDSSel ACCESS ADR(tyP1023McSetHComm.tyDSSel2);
			p_tyP1023McSetHCommDSSMEMA ACCESS ADR(tyP1023McSetHComm.tyDSSMEMA2);
			p_tyP1023McSetHCommDSHermes ACCESS ADR(tyP1023McSetHComm.tyDSHermes2);

			fUIInRtStatHide(ADR(tyP1023McSetHComm.tyDSSel.tyLyr.uiRtStat));
			fUIInRtStatOff(ADR(tyP1023McSetHComm.tyDSSel2.tyLyr.uiRtStat));

		END_IF

	ELSIF tyP1023McSetHComm.tyNaviLyr2.tyBtnLeft.bRtCompl = TRUE OR tyP1023McSetHComm.tyNaviLyr2.tyBtnRgt.bRtCompl = TRUE THEN
		tyP1023McSetHComm.tyNaviLyr2.tyBtnLeft.bRtCompl	:= FALSE;
		tyP1023McSetHComm.tyNaviLyr2.tyBtnRgt.bRtCompl	:= FALSE;

		p_tyC0004Navi ACCESS ADR(tyP1023McSetHComm.tyNaviLyr1);

		fUIInRtStatHide(ADR(tyP1023McSetHComm.tyDSSel.tyLyr.uiRtStat));
		fUIInRtStatHide(ADR(tyP1023McSetHComm.tyDSSel2.tyLyr.uiRtStat));

		IF tyP1023McSetHComm.tyGen.tyDrpDnUSSel.usiValueIdx = 0 THEN

			p_tyP1023McSetHCommUSSel ACCESS ADR(tyP1023McSetHComm.tyUSSel);
			p_tyP1023McSetHCommUSSMEMA ACCESS ADR(tyP1023McSetHComm.tyUSSMEMA);
			p_tyP1023McSetHCommUSHermes ACCESS ADR(tyP1023McSetHComm.tyUSHermes);

			fUIInRtStatOff(ADR(tyP1023McSetHComm.tyUSSel.tyLyr.uiRtStat));
			fUIInRtStatHide(ADR(tyP1023McSetHComm.tyUSSel2.tyLyr.uiRtStat));

		ELSIF tyP1023McSetHComm.tyGen.tyDrpDnUSSel.usiValueIdx = 1 THEN

			p_tyP1023McSetHCommUSSel ACCESS ADR(tyP1023McSetHComm.tyUSSel2);
			p_tyP1023McSetHCommUSSMEMA ACCESS ADR(tyP1023McSetHComm.tyUSSMEMA2);
			p_tyP1023McSetHCommUSHermes ACCESS ADR(tyP1023McSetHComm.tyUSHermes2);

			fUIInRtStatHide(ADR(tyP1023McSetHComm.tyUSSel.tyLyr.uiRtStat));
			fUIInRtStatOff(ADR(tyP1023McSetHComm.tyUSSel2.tyLyr.uiRtStat));

		END_IF

//Testing
//	ELSIF 	(tyP1023McSetHComm.tyNaviLyr2.tyBtnLeft.bRtCompl = TRUE OR tyP1023McSetHComm.tyNaviLyr2.tyBtnRgt.bRtCompl = TRUE) AND
//			tyP1023McSetHComm.tyGen.tyDrpDnUSSel.usiValueIdx = 0  THEN
//			tyP1023McSetHComm.tyNaviLyr2.tyBtnLeft.bRtCompl	:= FALSE;
//			tyP1023McSetHComm.tyNaviLyr2.tyBtnRgt.bRtCompl	:= FALSE;
//
//			p_tyC0004Navi ACCESS ADR(tyP1023McSetHComm.tyNaviLyr1);
//			p_tyP1023McSetHCommUSSel ACCESS ADR(tyP1023McSetHComm.tyUSSel);
//			p_tyP1023McSetHCommUSSMEMA ACCESS ADR(tyP1023McSetHComm.tyUSSMEMA);
//			p_tyP1023McSetHCommUSHermes ACCESS ADR(tyP1023McSetHComm.tyUSHermes);
//
//			fUIInRtStatHide(ADR(tyP1023McSetHComm.tyDSSel.tyLyr.uiRtStat));
//			fUIInRtStatOff(ADR(tyP1023McSetHComm.tyUSSel.tyLyr.uiRtStat));
//			fUIInRtStatHide(ADR(tyP1023McSetHComm.tyUSSel2.tyLyr.uiRtStat));
//
//	ELSIF 	(tyP1023McSetHComm.tyNaviLyr2.tyBtnLeft.bRtCompl = TRUE OR tyP1023McSetHComm.tyNaviLyr2.tyBtnRgt.bRtCompl = TRUE) AND
//			tyP1023McSetHComm.tyGen.tyDrpDnUSSel.usiValueIdx = 1 THEN
//			tyP1023McSetHComm.tyNaviLyr2.tyBtnLeft.bRtCompl	:= FALSE;
//			tyP1023McSetHComm.tyNaviLyr2.tyBtnRgt.bRtCompl	:= FALSE;
//
//			p_tyC0004Navi ACCESS ADR(tyP1023McSetHComm.tyNaviLyr1);
//			p_tyP1023McSetHCommUSSel ACCESS ADR(tyP1023McSetHComm.tyUSSel2);
//			p_tyP1023McSetHCommUSSMEMA ACCESS ADR(tyP1023McSetHComm.tyUSSMEMA2);
//
//			fUIInRtStatHide(ADR(tyP1023McSetHComm.tyDSSel.tyLyr.uiRtStat));
//			fUIInRtStatHide(ADR(tyP1023McSetHComm.tyUSSel.tyLyr.uiRtStat));
//			fUIInRtStatOff(ADR(tyP1023McSetHComm.tyUSSel2.tyLyr.uiRtStat));

	END_IF

END_ACTION
```

#### Act_OptP1023ShowLyr.st
```iecst
ACTION Act_OptP1023ShowLyr:

	IF tyP1023McSetHComm.tyUSSel.tyLyr.uiRtStat.0 = FALSE THEN
		fUIInRtStatHide(ADR(tyP1023McSetHComm.tyDSSMEMA.tyLyr.uiRtStat));
		fUIInRtStatHide(ADR(tyP1023McSetHComm.tyDSSMEMA2.tyLyr.uiRtStat));
		fUIInRtStatHide(ADR(tyP1023McSetHComm.tyDSHermes.tyLyr.uiRtStat));
		fUIInRtStatHide(ADR(tyP1023McSetHComm.tyDSHermes2.tyLyr.uiRtStat));
		fUIInRtStatHide(ADR(tyP1023McSetHComm.tyUSSMEMA2.tyLyr.uiRtStat));
		fUIInRtStatHide(ADR(tyP1023McSetHComm.tyUSHermes2.tyLyr.uiRtStat));

		IF tyP1023McSetHComm.tyUSSel.tyBtnSMEMA.bValue = TRUE THEN
			fUIInRtStatOff(ADR(tyP1023McSetHComm.tyUSSMEMA.tyLyr.uiRtStat));
			fUIInRtStatHide(ADR(tyP1023McSetHComm.tyUSHermes.tyLyr.uiRtStat));

			tyP1023McSetHComm.tyUSSMEMA.tyBtnGdSig.uiRtStat.0	:= NOT(tyP1023McSetHComm.tyUSSMEMA.tyDrpDnSMEMAMod.usiValueIdx = 2);

		ELSIF tyP1023McSetHComm.tyUSSel.tyBtnHermes.bValue = TRUE THEN
			fUIInRtStatHide(ADR(tyP1023McSetHComm.tyUSSMEMA.tyLyr.uiRtStat));
			fUIInRtStatOff(ADR(tyP1023McSetHComm.tyUSHermes.tyLyr.uiRtStat));

			//Mask
			tyP1023McSetHComm.tyUSHermes.tyBitmapMask.uiRtStat.0	:= NOT(p_tyNtParamCurr.bHermesRmtPrep = TRUE AND p_tyMcParamCurr.bHermesRmtEn = TRUE);
		END_IF

	ELSIF tyP1023McSetHComm.tyUSSel2.tyLyr.uiRtStat.0 = FALSE THEN
		fUIInRtStatHide(ADR(tyP1023McSetHComm.tyDSSMEMA.tyLyr.uiRtStat));
		fUIInRtStatHide(ADR(tyP1023McSetHComm.tyDSSMEMA2.tyLyr.uiRtStat));
		fUIInRtStatHide(ADR(tyP1023McSetHComm.tyDSHermes.tyLyr.uiRtStat));
		fUIInRtStatHide(ADR(tyP1023McSetHComm.tyDSHermes2.tyLyr.uiRtStat));
		fUIInRtStatHide(ADR(tyP1023McSetHComm.tyUSSMEMA.tyLyr.uiRtStat));
		fUIInRtStatHide(ADR(tyP1023McSetHComm.tyUSHermes.tyLyr.uiRtStat));

		IF tyP1023McSetHComm.tyUSSel2.tyBtnSMEMA.bValue = TRUE THEN
			fUIInRtStatOff(ADR(tyP1023McSetHComm.tyUSSMEMA2.tyLyr.uiRtStat));
			fUIInRtStatHide(ADR(tyP1023McSetHComm.tyUSHermes2.tyLyr.uiRtStat));

			tyP1023McSetHComm.tyUSSMEMA2.tyBtnGdSig.uiRtStat.0	:= NOT(tyP1023McSetHComm.tyUSSMEMA2.tyDrpDnSMEMAMod.usiValueIdx = 2);

		ELSIF tyP1023McSetHComm.tyUSSel2.tyBtnHermes.bValue = TRUE THEN
			fUIInRtStatHide(ADR(tyP1023McSetHComm.tyUSSMEMA2.tyLyr.uiRtStat));
			fUIInRtStatOff(ADR(tyP1023McSetHComm.tyUSHermes2.tyLyr.uiRtStat));

			//Mask
			tyP1023McSetHComm.tyUSHermes2.tyBitmapMask.uiRtStat.0	:= NOT(p_tyNtParamCurr.bHermesRmtPrep = TRUE AND p_tyMcParamCurr.bHermesRmtEn = TRUE);
		END_IF

	ELSIF tyP1023McSetHComm.tyDSSel.tyLyr.uiRtStat.0 = FALSE THEN
		fUIInRtStatHide(ADR(tyP1023McSetHComm.tyUSSMEMA.tyLyr.uiRtStat));
		fUIInRtStatHide(ADR(tyP1023McSetHComm.tyUSHermes.tyLyr.uiRtStat));
		fUIInRtStatHide(ADR(tyP1023McSetHComm.tyUSSMEMA2.tyLyr.uiRtStat));
		fUIInRtStatHide(ADR(tyP1023McSetHComm.tyUSHermes2.tyLyr.uiRtStat));
		fUIInRtStatHide(ADR(tyP1023McSetHComm.tyDSSMEMA2.tyLyr.uiRtStat));
		fUIInRtStatHide(ADR(tyP1023McSetHComm.tyDSHermes2.tyLyr.uiRtStat));

		IF tyP1023McSetHComm.tyDSSel.tyBtnSMEMA.bValue = TRUE THEN

			fUIInRtStatOff(ADR(tyP1023McSetHComm.tyDSSMEMA.tyLyr.uiRtStat));
			fUIInRtStatHide(ADR(tyP1023McSetHComm.tyDSHermes.tyLyr.uiRtStat));

			tyP1023McSetHComm.tyDSSMEMA.tyBtnGdSig.uiRtStat.0	:= NOT(tyP1023McSetHComm.tyDSSMEMA.tyDrpDnSMEMAMod.usiValueIdx = 2);

		ELSIF tyP1023McSetHComm.tyDSSel.tyBtnHermes.bValue = TRUE THEN

			fUIInRtStatHide(ADR(tyP1023McSetHComm.tyDSSMEMA.tyLyr.uiRtStat));
			fUIInRtStatOff(ADR(tyP1023McSetHComm.tyDSHermes.tyLyr.uiRtStat));

			//Mask
			tyP1023McSetHComm.tyDSHermes.tyBitmapMask.uiRtStat.0	:= NOT(p_tyNtParamCurr.bHermesRmtPrep = TRUE AND p_tyMcParamCurr.bHermesRmtEn = TRUE);
		END_IF
	ELSIF tyP1023McSetHComm.tyDSSel2.tyLyr.uiRtStat.0 = FALSE THEN
		fUIInRtStatHide(ADR(tyP1023McSetHComm.tyUSSMEMA.tyLyr.uiRtStat));
		fUIInRtStatHide(ADR(tyP1023McSetHComm.tyUSHermes.tyLyr.uiRtStat));
		fUIInRtStatHide(ADR(tyP1023McSetHComm.tyUSSMEMA2.tyLyr.uiRtStat));
		fUIInRtStatHide(ADR(tyP1023McSetHComm.tyUSHermes2.tyLyr.uiRtStat));
		fUIInRtStatHide(ADR(tyP1023McSetHComm.tyDSSMEMA.tyLyr.uiRtStat));
		fUIInRtStatHide(ADR(tyP1023McSetHComm.tyDSHermes.tyLyr.uiRtStat));

		IF tyP1023McSetHComm.tyDSSel2.tyBtnSMEMA.bValue = TRUE THEN
			fUIInRtStatOff(ADR(tyP1023McSetHComm.tyDSSMEMA2.tyLyr.uiRtStat));
			fUIInRtStatHide(ADR(tyP1023McSetHComm.tyDSHermes2.tyLyr.uiRtStat));

			tyP1023McSetHComm.tyDSSMEMA2.tyBtnGdSig.uiRtStat.0	:= NOT(tyP1023McSetHComm.tyDSSMEMA2.tyDrpDnSMEMAMod.usiValueIdx = 2);

		ELSIF tyP1023McSetHComm.tyDSSel2.tyBtnHermes.bValue = TRUE THEN
			fUIInRtStatHide(ADR(tyP1023McSetHComm.tyDSSMEMA2.tyLyr.uiRtStat));
			fUIInRtStatOff(ADR(tyP1023McSetHComm.tyDSHermes2.tyLyr.uiRtStat));

			//Mask
			tyP1023McSetHComm.tyDSHermes2.tyBitmapMask.uiRtStat.0	:= NOT(p_tyNtParamCurr.bHermesRmtPrep = TRUE AND p_tyMcParamCurr.bHermesRmtEn = TRUE);
		END_IF
	ELSE

		fUIInRtStatHide(ADR(tyP1023McSetHComm.tyUSSMEMA.tyLyr.uiRtStat));
		fUIInRtStatHide(ADR(tyP1023McSetHComm.tyUSHermes.tyLyr.uiRtStat));
		fUIInRtStatHide(ADR(tyP1023McSetHComm.tyUSSMEMA2.tyLyr.uiRtStat));
		fUIInRtStatHide(ADR(tyP1023McSetHComm.tyUSHermes2.tyLyr.uiRtStat));
		fUIInRtStatHide(ADR(tyP1023McSetHComm.tyDSSMEMA.tyLyr.uiRtStat));
		fUIInRtStatHide(ADR(tyP1023McSetHComm.tyDSHermes.tyLyr.uiRtStat));
		fUIInRtStatHide(ADR(tyP1023McSetHComm.tyDSSMEMA2.tyLyr.uiRtStat));
		fUIInRtStatHide(ADR(tyP1023McSetHComm.tyDSHermes2.tyLyr.uiRtStat));
	END_IF

END_ACTION
```

#### Act_OptP1023Save.st
```iecst
ACTION Act_OptP1023Save:

	IF tyP1023McSetHComm.tyUSSel.tyBtnSMEMA.bRtCompl						OR tyP1023McSetHComm.tyUSSel.tyBtnHermes.bRtCompl
		OR tyP1023McSetHComm.tyUSSMEMA.tyDrpDnSMEMAMod.bRtCompl				OR tyP1023McSetHComm.tyUSSMEMA.tyBtnGdSig.bRtCompl
		OR tyP1023McSetHComm.tyUSHermes.tyNumSndAliveTm.bRtCompl			OR tyP1023McSetHComm.tyUSHermes.tyNumLaneID.bRtCompl
		OR tyP1023McSetHComm.tyUSHermes.tyStringHostAddr.bRtCompl			OR tyP1023McSetHComm.tyUSHermes.tyNumHostPort.bRtCompl
		OR tyP1023McSetHComm.tyUSHermes.tyBtnCheckAliveResponse.bRtCompl	OR tyP1023McSetHComm.tyUSHermes.tyBtnCmpTypeId.bRtCompl
		OR tyP1023McSetHComm.tyUSHermes.tyBtnCmpParam.bRtCompl				OR tyP1023McSetHComm.tyUSHermes.tyBtnOverWrite.bRtCompl
		OR tyP1023McSetHComm.tyUSHermes.tyBtnBoardForecast.bRtCompl		OR tyP1023McSetHComm.tyUSHermes.tyBtnQueryBoardInfo.bRtCompl
		OR tyP1023McSetHComm.tyUSHermes.tyBtnCommand.bRtCompl

		OR tyP1023McSetHComm.tyUSSel2.tyBtnSMEMA.bRtCompl					OR tyP1023McSetHComm.tyUSSel2.tyBtnHermes.bRtCompl
		OR tyP1023McSetHComm.tyUSSMEMA2.tyDrpDnSMEMAMod.bRtCompl			OR tyP1023McSetHComm.tyUSSMEMA2.tyBtnGdSig.bRtCompl

		OR tyP1023McSetHComm.tyDSSel.tyBtnSMEMA.bRtCompl					OR tyP1023McSetHComm.tyDSSel.tyBtnHermes.bRtCompl
		OR tyP1023McSetHComm.tyDSSMEMA.tyDrpDnSMEMAMod.bRtCompl				OR tyP1023McSetHComm.tyDSSMEMA.tyBtnGdSig.bRtCompl
		OR tyP1023McSetHComm.tyDSHermes.tyNumSndAliveTm.bRtCompl			OR tyP1023McSetHComm.tyDSHermes.tyNumLaneID.bRtCompl
		OR tyP1023McSetHComm.tyDSHermes.tyNumSvrPort.bRtCompl				OR tyP1023McSetHComm.tyDSHermes.tyBtnCheckAliveResponse.bRtCompl
		OR tyP1023McSetHComm.tyDSHermes.tyBtnBoardForecast.bRtCompl			OR tyP1023McSetHComm.tyDSHermes.tyBtnSendBoardInfo.bRtCompl
		OR tyP1023McSetHComm.tyDSHermes.tyBtnCommand.bRtCompl

		OR tyP1023McSetHComm.tyUSHermes2.tyNumSndAliveTm.bRtCompl			OR tyP1023McSetHComm.tyUSHermes2.tyNumLaneID.bRtCompl
		OR tyP1023McSetHComm.tyUSHermes2.tyStringHostAddr.bRtCompl			OR tyP1023McSetHComm.tyUSHermes2.tyNumHostPort.bRtCompl
		OR tyP1023McSetHComm.tyUSHermes2.tyBtnCheckAliveResponse.bRtCompl	OR tyP1023McSetHComm.tyUSHermes2.tyBtnCmpTypeId.bRtCompl
		OR tyP1023McSetHComm.tyUSHermes2.tyBtnCmpParam.bRtCompl				OR tyP1023McSetHComm.tyUSHermes2.tyBtnOverWrite.bRtCompl
		OR tyP1023McSetHComm.tyUSHermes2.tyBtnBoardForecast.bRtCompl		OR tyP1023McSetHComm.tyUSHermes2.tyBtnQueryBoardInfo.bRtCompl
		OR tyP1023McSetHComm.tyUSHermes2.tyBtnCommand.bRtCompl  //Hermes2

		OR tyP1023McSetHComm.tyDSSel2.tyBtnSMEMA.bRtCompl					OR tyP1023McSetHComm.tyDSSel2.tyBtnHermes.bRtCompl
		OR tyP1023McSetHComm.tyDSSMEMA2.tyDrpDnSMEMAMod.bRtCompl			OR tyP1023McSetHComm.tyDSSMEMA2.tyBtnGdSig.bRtCompl
		OR tyP1023McSetHComm.tyDSHermes2.tyNumSndAliveTm.bRtCompl			OR tyP1023McSetHComm.tyDSHermes2.tyNumLaneID.bRtCompl
		OR tyP1023McSetHComm.tyDSHermes2.tyNumSvrPort.bRtCompl				OR tyP1023McSetHComm.tyDSHermes2.tyBtnCheckAliveResponse.bRtCompl
		OR tyP1023McSetHComm.tyDSHermes2.tyBtnBoardForecast.bRtCompl		OR tyP1023McSetHComm.tyDSHermes2.tyBtnSendBoardInfo.bRtCompl
		OR tyP1023McSetHComm.tyDSHermes2.tyBtnCommand.bRtCompl

		THEN

		fUIInRtStatHide(ADR(tyCommon.tySet.tyBtnSave.uiMaskRtStat));

		tyP1023McSetHComm.tyUSSMEMA.tyDrpDnSMEMAMod.bRtCompl			:= FALSE;
		tyP1023McSetHComm.tyUSSMEMA.tyBtnGdSig.bRtCompl					:= FALSE;
		tyP1023McSetHComm.tyUSHermes.tyNumSndAliveTm.bRtCompl			:= FALSE;
		tyP1023McSetHComm.tyUSHermes.tyNumLaneID.bRtCompl				:= FALSE;
		tyP1023McSetHComm.tyUSHermes.tyStringHostAddr.bRtCompl			:= FALSE;
		tyP1023McSetHComm.tyUSHermes.tyNumHostPort.bRtCompl				:= FALSE;
		tyP1023McSetHComm.tyUSHermes.tyBtnCheckAliveResponse.bRtCompl	:= FALSE;
		tyP1023McSetHComm.tyUSHermes.tyBtnCmpTypeId.bRtCompl			:= FALSE;
		tyP1023McSetHComm.tyUSHermes.tyBtnCmpParam.bRtCompl				:= FALSE;
		tyP1023McSetHComm.tyUSHermes.tyBtnOverWrite.bRtCompl			:= FALSE;
		tyP1023McSetHComm.tyUSHermes.tyBtnBoardForecast.bRtCompl		:= FALSE;
		tyP1023McSetHComm.tyUSHermes.tyBtnQueryBoardInfo.bRtCompl		:= FALSE;
		tyP1023McSetHComm.tyUSHermes.tyBtnCommand.bRtCompl				:= FALSE;

		tyP1023McSetHComm.tyUSSMEMA2.tyDrpDnSMEMAMod.bRtCompl			:= FALSE;
		tyP1023McSetHComm.tyUSSMEMA2.tyBtnGdSig.bRtCompl				:= FALSE;

		tyP1023McSetHComm.tyDSSMEMA.tyDrpDnSMEMAMod.bRtCompl			:= FALSE;
		tyP1023McSetHComm.tyDSSMEMA.tyBtnGdSig.bRtCompl					:= FALSE;
		tyP1023McSetHComm.tyDSHermes.tyNumSndAliveTm.bRtCompl			:= FALSE;
		tyP1023McSetHComm.tyDSHermes.tyNumLaneID.bRtCompl				:= FALSE;
		tyP1023McSetHComm.tyDSHermes.tyNumSvrPort.bRtCompl				:= FALSE;
		tyP1023McSetHComm.tyDSHermes.tyBtnCheckAliveResponse.bRtCompl	:= FALSE;
		tyP1023McSetHComm.tyDSHermes.tyBtnBoardForecast.bRtCompl		:= FALSE;
		tyP1023McSetHComm.tyDSHermes.tyBtnSendBoardInfo.bRtCompl		:= FALSE;
		tyP1023McSetHComm.tyDSHermes.tyBtnCommand.bRtCompl				:= FALSE;

		tyP1023McSetHComm.tyUSHermes2.tyNumSndAliveTm.bRtCompl			:= FALSE;
		tyP1023McSetHComm.tyUSHermes2.tyNumLaneID.bRtCompl				:= FALSE;
		tyP1023McSetHComm.tyUSHermes2.tyStringHostAddr.bRtCompl			:= FALSE;
		tyP1023McSetHComm.tyUSHermes2.tyNumHostPort.bRtCompl			:= FALSE;
		tyP1023McSetHComm.tyUSHermes2.tyBtnCheckAliveResponse.bRtCompl	:= FALSE;
		tyP1023McSetHComm.tyUSHermes2.tyBtnCmpTypeId.bRtCompl			:= FALSE;
		tyP1023McSetHComm.tyUSHermes2.tyBtnCmpParam.bRtCompl			:= FALSE;
		tyP1023McSetHComm.tyUSHermes2.tyBtnOverWrite.bRtCompl			:= FALSE;
		tyP1023McSetHComm.tyUSHermes2.tyBtnBoardForecast.bRtCompl		:= FALSE;
		tyP1023McSetHComm.tyUSHermes2.tyBtnQueryBoardInfo.bRtCompl		:= FALSE;
		tyP1023McSetHComm.tyUSHermes2.tyBtnCommand.bRtCompl				:= FALSE;

		//DS SMEMA 2 and Hermes2

		tyP1023McSetHComm.tyDSSMEMA2.tyDrpDnSMEMAMod.bRtCompl			:= FALSE;
		tyP1023McSetHComm.tyDSSMEMA2.tyBtnGdSig.bRtCompl				:= FALSE;
		tyP1023McSetHComm.tyDSHermes2.tyNumSndAliveTm.bRtCompl			:= FALSE;
		tyP1023McSetHComm.tyDSHermes2.tyNumLaneID.bRtCompl				:= FALSE;
		tyP1023McSetHComm.tyDSHermes2.tyNumSvrPort.bRtCompl				:= FALSE;
		tyP1023McSetHComm.tyDSHermes2.tyBtnCheckAliveResponse.bRtCompl	:= FALSE;
		tyP1023McSetHComm.tyDSHermes2.tyBtnBoardForecast.bRtCompl		:= FALSE;
		tyP1023McSetHComm.tyDSHermes2.tyBtnSendBoardInfo.bRtCompl		:= FALSE;
		tyP1023McSetHComm.tyDSHermes2.tyBtnCommand.bRtCompl				:= FALSE;

	END_IF

	IF tyCommon.tySet.tyBtnSave.bRtCompl = TRUE THEN
		IF usiSaveCommStep = 0 THEN
			//Verify IP Address
			IF (tyP1023McSetHComm.tyUSSel.tyBtnHermes.bValue = TRUE) AND NOT(p_tyNtParamCurr.bHermesRmtPrep = TRUE AND p_tyMcParamCurr.bHermesRmtEn = TRUE) THEN
				IF fIPValid(tyP1023McSetHComm.tyUSHermes.tyStringHostAddr.sValue, ADR(a_iIPPart1)) = TRUE THEN
					usiSaveCommStep	:= 1;
				ELSE
					usiSaveCommStep	:= 99;
				END_IF
			ELSE
				usiSaveCommStep	:= 1;
			END_IF

		ELSIF usiSaveCommStep = 1 THEN
			//Save Machine Parameter
			//Upstream
			IF tyP1023McSetHComm.tyUSSel.tyBtnSMEMA.bValue = TRUE THEN
				tyMcParamWr.eUSComm	:= McSetCommModSMEMA;
			ELSIF tyP1023McSetHComm.tyUSSel.tyBtnHermes.bValue = TRUE THEN
				tyMcParamWr.eUSComm	:= McSetCommModHermes;
			END_IF

			tyMcParamWr.tyUSCommSMEMA.eSelection	:= USINT_TO_UDINT(tyP1023McSetHComm.tyUSSMEMA.tyDrpDnSMEMAMod.usiValueIdx);
			tyMcParamWr.tyUSCommSMEMA.bStatSigSetGd	:= tyP1023McSetHComm.tyUSSMEMA.tyBtnGdSig.bValue;

			//Upstream 2
			IF tyP1023McSetHComm.tyUSSel2.tyBtnSMEMA.bValue = TRUE THEN
				tyMcParamWr.eUSComm2	:= McSetCommModSMEMA;
			ELSIF tyP1023McSetHComm.tyUSSel2.tyBtnHermes.bValue = TRUE THEN
				tyMcParamWr.eUSComm2	:= McSetCommModHermes;
			END_IF

			tyMcParamWr.tyUSCommSMEMA2.eSelection		:= USINT_TO_UDINT(tyP1023McSetHComm.tyUSSMEMA2.tyDrpDnSMEMAMod.usiValueIdx);
			tyMcParamWr.tyUSCommSMEMA2.bStatSigSetGd	:= tyP1023McSetHComm.tyUSSMEMA2.tyBtnGdSig.bValue;

			//Downstream
			IF tyP1023McSetHComm.tyDSSel.tyBtnSMEMA.bValue = TRUE THEN
				tyMcParamWr.eDSComm	:= McSetCommModSMEMA;
			ELSIF tyP1023McSetHComm.tyDSSel.tyBtnHermes.bValue = TRUE THEN
				tyMcParamWr.eDSComm	:= McSetCommModHermes;
			END_IF

			tyMcParamWr.tyDSCommSMEMA.eSelection	:= USINT_TO_UDINT(tyP1023McSetHComm.tyDSSMEMA.tyDrpDnSMEMAMod.usiValueIdx);
			tyMcParamWr.tyDSCommSMEMA.bStatSigSetGd	:= tyP1023McSetHComm.tyDSSMEMA.tyBtnGdSig.bValue;

			//Downstream
			IF tyP1023McSetHComm.tyDSSel2.tyBtnSMEMA.bValue = TRUE THEN
				tyMcParamWr.eDSComm2	:= McSetCommModSMEMA;
			ELSIF tyP1023McSetHComm.tyDSSel2.tyBtnHermes.bValue = TRUE THEN
				tyMcParamWr.eDSComm2	:= McSetCommModHermes;
			END_IF

			tyMcParamWr.tyDSCommSMEMA2.eSelection	:= USINT_TO_UDINT(tyP1023McSetHComm.tyDSSMEMA2.tyDrpDnSMEMAMod.usiValueIdx);
			tyMcParamWr.tyDSCommSMEMA2.bStatSigSetGd	:= tyP1023McSetHComm.tyDSSMEMA2.tyBtnGdSig.bValue;

			eMcParamAct	:= McParamActWrite;

			IF p_eMcParamStat = McParamActWrite AND p_eMcParamStatus = Done THEN
				eMcParamAct	:= McParamActIdle;

				//Backup Param
				tyP1023McSetHComm.tyUSSelBkUp		:= tyP1023McSetHComm.tyUSSel;
				tyP1023McSetHComm.tyUSSMEMABkUp		:= tyP1023McSetHComm.tyUSSMEMA;
				tyP1023McSetHComm.tyDSSelBkUp		:= tyP1023McSetHComm.tyDSSel;
				tyP1023McSetHComm.tyDSSMEMABkUp		:= tyP1023McSetHComm.tyDSSMEMA;
				tyP1023McSetHComm.tyUSSelBkUp2		:= tyP1023McSetHComm.tyUSSel2;
				tyP1023McSetHComm.tyUSSMEMABkUp2	:= tyP1023McSetHComm.tyUSSMEMA2;

				usiSaveCommStep	:= 2;

			ELSIF p_eMcParamStatus = Error THEN
				p_tyC0008MsgBox ACCESS ADR(tyP1023McSetHComm.tyMsgBoxSaveErr);

				IF tyP1023McSetHComm.tyMsgBoxSaveErr.tyBtnNo.bRtCompl = TRUE THEN
					tyP1023McSetHComm.tyMsgBoxSaveErr.tyBtnNo.bRtCompl	:= FALSE;
					tyP1023McSetHComm.tyMsgBoxSaveErr.tyBtnNo.bValue	:= FALSE;

					p_tyC0008MsgBox ACCESS ADR(tyP1023McSetHComm.tyMsgBoxHide);

					//Restore Param
					tyP1023McSetHComm.tyUSSel		:= tyP1023McSetHComm.tyUSSelBkUp;
					tyP1023McSetHComm.tyUSSMEMA		:= tyP1023McSetHComm.tyUSSMEMABkUp;
					tyP1023McSetHComm.tyDSSel		:= tyP1023McSetHComm.tyDSSelBkUp;
					tyP1023McSetHComm.tyDSSMEMA		:= tyP1023McSetHComm.tyDSSMEMABkUp;
					tyP1023McSetHComm.tyUSSel2		:= tyP1023McSetHComm.tyUSSelBkUp2;
					tyP1023McSetHComm.tyUSSMEMA2	:= tyP1023McSetHComm.tyUSSMEMABkUp2;

					tyMcParamWr					:= p_tyMcParamCurr;

					usiSaveCommStep	:= 2;

				END_IF

			END_IF

		ELSIF usiSaveCommStep = 2 THEN
			//Save Hermes Configuration
			//Upstream
			a_tyHermesUSParamWr[0].tSndAlive					:= DINT_TO_TIME(tyP1023McSetHComm.tyUSHermes.tyNumSndAliveTm.diValue);
			a_tyHermesUSParamWr[0].iLaneID						:= DINT_TO_INT(tyP1023McSetHComm.tyUSHermes.tyNumLaneID.diValue);
			a_tyHermesUSParamWr[0].uiHostPort					:= DINT_TO_UINT(tyP1023McSetHComm.tyUSHermes.tyNumHostPort.diValue);
			a_tyHermesUSParamWr[0].sHostAddress					:= tyP1023McSetHComm.tyUSHermes.tyStringHostAddr.sValue;
			a_tyHermesUSParamWr[0].bFeatureCheckAliveResponse	:= tyP1023McSetHComm.tyUSHermes.tyBtnCheckAliveResponse.bValue;
			a_tyHermesUSParamWr[0].bFeatureBoardForecast		:= tyP1023McSetHComm.tyUSHermes.tyBtnBoardForecast.bValue;
			a_tyHermesUSParamWr[0].bFeatureQueryBoardInfo		:= tyP1023McSetHComm.tyUSHermes.tyBtnQueryBoardInfo.bValue;
			a_tyHermesUSParamWr[0].bFeatureCommand				:= tyP1023McSetHComm.tyUSHermes.tyBtnCommand.bValue;
			a_tyHermesUSParamWr[0].bCmpTypeId					:= tyP1023McSetHComm.tyUSHermes.tyBtnCmpTypeId.bValue;
			a_tyHermesUSParamWr[0].bCmpParam					:= tyP1023McSetHComm.tyUSHermes.tyBtnCmpParam.bValue;
			a_tyHermesUSParamWr[0].bOverwrite					:= tyP1023McSetHComm.tyUSHermes.tyBtnOverWrite.bValue;

			//Upstream 2
			a_tyHermesUSParamWr[1].tSndAlive					:= DINT_TO_TIME(tyP1023McSetHComm.tyUSHermes2.tyNumSndAliveTm.diValue);
			a_tyHermesUSParamWr[1].iLaneID						:= DINT_TO_INT(tyP1023McSetHComm.tyUSHermes2.tyNumLaneID.diValue);
			a_tyHermesUSParamWr[1].uiHostPort					:= DINT_TO_UINT(tyP1023McSetHComm.tyUSHermes2.tyNumHostPort.diValue);
			a_tyHermesUSParamWr[1].sHostAddress					:= tyP1023McSetHComm.tyUSHermes2.tyStringHostAddr.sValue;
			a_tyHermesUSParamWr[1].bFeatureCheckAliveResponse	:= tyP1023McSetHComm.tyUSHermes2.tyBtnCheckAliveResponse.bValue;
			a_tyHermesUSParamWr[1].bFeatureBoardForecast		:= tyP1023McSetHComm.tyUSHermes2.tyBtnBoardForecast.bValue;
			a_tyHermesUSParamWr[1].bFeatureQueryBoardInfo		:= tyP1023McSetHComm.tyUSHermes2.tyBtnQueryBoardInfo.bValue;
			a_tyHermesUSParamWr[1].bFeatureCommand				:= tyP1023McSetHComm.tyUSHermes2.tyBtnCommand.bValue;
			a_tyHermesUSParamWr[1].bCmpTypeId					:= tyP1023McSetHComm.tyUSHermes2.tyBtnCmpTypeId.bValue;
			a_tyHermesUSParamWr[1].bCmpParam					:= tyP1023McSetHComm.tyUSHermes2.tyBtnCmpParam.bValue;
			a_tyHermesUSParamWr[1].bOverwrite					:= tyP1023McSetHComm.tyUSHermes2.tyBtnOverWrite.bValue;

			//Downstream
			a_tyHermesDSParamWr[0].tSndAlive					:= DINT_TO_TIME(tyP1023McSetHComm.tyDSHermes.tyNumSndAliveTm.diValue);
			a_tyHermesDSParamWr[0].uiSvrPort					:= DINT_TO_UINT(tyP1023McSetHComm.tyDSHermes.tyNumSvrPort.diValue);
			a_tyHermesDSParamWr[0].iLaneID						:= DINT_TO_INT(tyP1023McSetHComm.tyDSHermes.tyNumLaneID.diValue);
			a_tyHermesDSParamWr[0].bFeatureCheckAliveResponse	:= tyP1023McSetHComm.tyDSHermes.tyBtnCheckAliveResponse.bValue;
			a_tyHermesDSParamWr[0].bFeatureBoardForecast	    := tyP1023McSetHComm.tyDSHermes.tyBtnBoardForecast.bValue;
			a_tyHermesDSParamWr[0].bFeatureSendBoardInfo    	:= tyP1023McSetHComm.tyDSHermes.tyBtnSendBoardInfo.bValue;
			a_tyHermesDSParamWr[0].bFeatureCommand				:= tyP1023McSetHComm.tyDSHermes.tyBtnCommand.bValue;

			//Downstream
			a_tyHermesDSParamWr[1].tSndAlive					:= DINT_TO_TIME(tyP1023McSetHComm.tyDSHermes2.tyNumSndAliveTm.diValue);
			a_tyHermesDSParamWr[1].uiSvrPort					:= DINT_TO_UINT(tyP1023McSetHComm.tyDSHermes2.tyNumSvrPort.diValue);
			a_tyHermesDSParamWr[1].iLaneID						:= DINT_TO_INT(tyP1023McSetHComm.tyDSHermes2.tyNumLaneID.diValue);
			a_tyHermesDSParamWr[1].bFeatureCheckAliveResponse	:= tyP1023McSetHComm.tyDSHermes2.tyBtnCheckAliveResponse.bValue;
			a_tyHermesDSParamWr[1].bFeatureBoardForecast	    := tyP1023McSetHComm.tyDSHermes2.tyBtnBoardForecast.bValue;
			a_tyHermesDSParamWr[1].bFeatureSendBoardInfo    	:= tyP1023McSetHComm.tyDSHermes2.tyBtnSendBoardInfo.bValue;
			a_tyHermesDSParamWr[1].bFeatureCommand				:= tyP1023McSetHComm.tyDSHermes2.tyBtnCommand.bValue;

			bSaveHMIConfigure := TRUE;
			eHermesAct	:= HermesActWriteConfig;

			IF p_eHermesStat = HermesActWriteConfig AND p_eHermesStatus = Done THEN
				eHermesAct	:= HermesActIdle;

				//Backup Param
				tyP1023McSetHComm.tyUSHermesBkUp	:= tyP1023McSetHComm.tyUSHermes;
				tyP1023McSetHComm.tyUSHermesBkUp2	:= tyP1023McSetHComm.tyUSHermes2;
				tyP1023McSetHComm.tyDSHermesBkUp	:= tyP1023McSetHComm.tyDSHermes;
				tyP1023McSetHComm.tyDSHermesBkUp2	:= tyP1023McSetHComm.tyDSHermes2;

				usiSaveCommStep	:= 0;
				bSaveHMIConfigure := FALSE;
				tyCommon.tySet.tyBtnSave.bRtCompl	:= FALSE;

				fUIInRtStatOff(ADR(tyCommon.tySet.tyBtnSave.uiMaskRtStat));

			ELSIF p_eHermesStatus = Error THEN
				p_tyC0008MsgBox ACCESS ADR(tyP1023McSetHComm.tyMsgBoxSaveErr);

				IF tyP1023McSetHComm.tyMsgBoxSaveErr.tyBtnNo.bRtCompl = TRUE THEN
					tyP1023McSetHComm.tyMsgBoxSaveErr.tyBtnNo.bRtCompl	:= FALSE;
					tyP1023McSetHComm.tyMsgBoxSaveErr.tyBtnNo.bValue	:= FALSE;

					p_tyC0008MsgBox ACCESS ADR(tyP1023McSetHComm.tyMsgBoxHide);

					//Restore Param
					tyP1023McSetHComm.tyUSHermes	:= tyP1023McSetHComm.tyUSHermesBkUp;
					tyP1023McSetHComm.tyUSHermes2	:= tyP1023McSetHComm.tyUSHermesBkUp2;
					tyP1023McSetHComm.tyDSHermes	:= tyP1023McSetHComm.tyDSHermesBkUp;
					tyP1023McSetHComm.tyDSHermes2	:= tyP1023McSetHComm.tyDSHermesBkUp2;

					a_tyHermesUSParamWr				:= p_tyHermesConfiguration.a_tyUSParam;
					a_tyHermesDSParamWr				:= p_tyHermesConfiguration.a_tyDSParam;

					tyCommon.tySet.tyBtnSave.bRtCompl	:= FALSE;
					bSaveHMIConfigure := FALSE;
					fUIInRtStatOff(ADR(tyCommon.tySet.tyBtnSave.uiMaskRtStat));

					usiSaveCommStep	:= 0;

				END_IF

			END_IF

		ELSIF usiSaveCommStep = 99 THEN
			p_tyC0008MsgBox ACCESS ADR(tyP1023McSetHComm.tyMsgBoxIPAddrInvalid);

			IF tyP1023McSetHComm.tyMsgBoxIPAddrInvalid.tyBtnNo.bRtCompl = TRUE THEN
				tyP1023McSetHComm.tyMsgBoxIPAddrInvalid.tyBtnNo.bRtCompl	:= FALSE;
				tyP1023McSetHComm.tyMsgBoxIPAddrInvalid.tyBtnNo.bValue		:= FALSE;

				p_tyC0008MsgBox ACCESS ADR(tyP1023McSetHComm.tyMsgBoxHide);

				//Restore Param
				tyP1023McSetHComm.tyUSSel		:= tyP1023McSetHComm.tyUSSelBkUp;
				tyP1023McSetHComm.tyUSSMEMA		:= tyP1023McSetHComm.tyUSSMEMABkUp;
				tyP1023McSetHComm.tyUSHermes	:= tyP1023McSetHComm.tyUSHermesBkUp;
				tyP1023McSetHComm.tyDSSel		:= tyP1023McSetHComm.tyDSSelBkUp;
				tyP1023McSetHComm.tyDSSMEMA		:= tyP1023McSetHComm.tyDSSMEMABkUp;
				tyP1023McSetHComm.tyDSHermes	:= tyP1023McSetHComm.tyDSHermesBkUp;
				tyP1023McSetHComm.tyUSSel2		:= tyP1023McSetHComm.tyUSSelBkUp2;
				tyP1023McSetHComm.tyUSSMEMA2	:= tyP1023McSetHComm.tyUSSMEMABkUp2;
				tyP1023McSetHComm.tyUSHermes2	:= tyP1023McSetHComm.tyUSHermesBkUp2;
				tyP1023McSetHComm.tyDSSel2		:= tyP1023McSetHComm.tyDSSelBkUp;
				tyP1023McSetHComm.tyDSSMEMA2		:= tyP1023McSetHComm.tyDSSMEMABkUp;
				tyP1023McSetHComm.tyDSHermes2	:= tyP1023McSetHComm.tyDSHermesBkUp;

				tyCommon.tySet.tyBtnSave.bRtCompl	:= FALSE;

				fUIInRtStatOff(ADR(tyCommon.tySet.tyBtnSave.uiMaskRtStat));

				usiSaveCommStep	:= 0;

			END_IF

		END_IF

	END_IF

END_ACTION
```
